C05450=1092.796,439.335,-104.729,178.655,25.944,154.047
C05451=1092.802,439.581,-104.773,178.657,25.957,154.050
C05452=1092.809,439.827,-104.817,178.661,25.970,154.053
C05453=1092.815,440.073,-104.861,178.665,25.983,154.056
C05454=1092.822,440.320,-104.905,178.667,25.995,154.059
C05455=1092.829,440.565,-104.948,178.671,26.009,154.062
C05456=1092.836,440.811,-104.992,178.674,26.022,154.065
C05457=1092.842,441.057,-105.036,178.677,26.035,154.068
C05458=1092.849,441.303,-105.080,178.680,26.048,154.071
C05459=1092.855,441.549,-105.124,178.684,26.061,154.074
C05460=1092.862,441.795,-105.168,178.687,26.074,154.077
C05461=1092.868,442.041,-105.212,178.690,26.088,154.080
C05462=1092.875,442.287,-105.256,178.693,26.101,154.083
C05463=1092.881,442.532,-105.299,178.697,26.115,154.086
C05464=1092.888,442.778,-105.344,178.700,26.128,154.089
C05465=1092.894,443.024,-105.388,178.703,26.142,154.092
C05466=1092.901,443.270,-105.432,178.707,26.155,154.095
C05467=1092.908,443.516,-105.477,178.710,26.169,154.098
C05468=1092.914,443.762,-105.521,178.713,26.182,154.101
C05469=1092.921,444.007,-105.565,178.716,26.196,154.104
C05470=1092.927,444.253,-105.610,178.719,26.210,154.107
C05471=1092.934,444.499,-105.654,178.723,26.224,154.110
C05472=1092.941,444.745,-105.698,178.725,26.237,154.114
C05473=1092.947,444.991,-105.743,178.728,26.251,154.117
C05474=1092.954,445.237,-105.787,178.730,26.265,154.120
C05475=1092.960,445.482,-105.831,178.733,26.279,154.123
C05476=1092.968,445.728,-105.876,178.735,26.292,154.126
C05477=1092.973,445.974,-105.921,178.737,26.306,154.130
C05478=1092.980,446.220,-105.965,178.738,26.319,154.133
C05479=1092.988,446.466,-106.010,178.741,26.333,154.136
C05480=1092.994,446.712,-106.054,178.741,26.347,154.140
C05481=1093.000,446.958,-106.099,178.743,26.361,154.143
C05482=1093.007,447.204,-106.144,178.744,26.374,154.146
C05483=1093.014,447.449,-106.189,178.745,26.388,154.150
C05484=1093.020,447.695,-106.233,178.746,26.401,154.153
C05485=1093.027,447.941,-106.278,178.747,26.415,154.156
C05486=1093.034,448.187,-106.323,178.747,26.429,154.160
C05487=1093.040,448.432,-106.368,178.747,26.442,154.163
C05488=1093.047,448.678,-106.413,178.748,26.456,154.166
C05489=1093.054,448.924,-106.457,178.748,26.469,154.170
C05490=1093.060,449.170,-106.503,178.748,26.483,154.173
C05491=1093.067,449.415,-106.547,178.747,26.496,154.177
C05492=1093.074,449.661,-106.592,178.748,26.510,154.180
C05493=1093.081,449.906,-106.637,178.748,26.523,154.184
C05494=1093.089,450.153,-106.681,178.747,26.535,154.187
C05495=1092.703,450.144,-106.858,178.697,26.740,154.244
C05496=1092.694,449.897,-106.813,178.697,26.727,154.241
C05497=1092.687,449.651,-106.768,178.698,26.714,154.237
C05498=1092.680,449.406,-106.724,178.698,26.700,154.234
C05499=1092.673,449.161,-106.679,178.698,26.686,154.230
C05500=1092.667,448.915,-106.634,178.698,26.673,154.227
C05501=1092.660,448.669,-106.589,178.698,26.660,154.224
C05502=1092.653,448.423,-106.544,178.697,26.646,154.220
C05503=1092.647,448.177,-106.499,178.697,26.633,154.217
C05504=1092.640,447.932,-106.454,178.697,26.619,154.213
C05505=1092.633,447.686,-106.409,178.695,26.605,154.210
C05506=1092.627,447.440,-106.364,178.695,26.591,154.207
C05507=1092.620,447.195,-106.320,178.694,26.578,154.203
C05508=1092.613,446.949,-106.275,178.692,26.564,154.200
C05509=1092.607,446.702,-106.230,178.691,26.550,154.197
C05510=1092.600,446.457,-106.186,178.689,26.536,154.193
C05511=1092.593,446.211,-106.141,178.687,26.523,154.190
C05512=1092.586,445.966,-106.096,178.686,26.509,154.187
C05513=1092.580,445.719,-106.052,178.684,26.495,154.183
C05514=1092.573,445.473,-106.007,178.682,26.482,154.180
C05515=1092.566,445.228,-105.962,178.679,26.468,154.177
C05516=1092.560,444.982,-105.918,178.677,26.454,154.174
C05517=1092.553,444.736,-105.874,178.674,26.440,154.170
C05518=1092.547,444.490,-105.828,178.671,26.427,154.167
C05519=1092.540,444.244,-105.785,178.668,26.413,154.164
C05520=1092.533,443.999,-105.740,178.664,26.399,154.161
C05521=1092.526,443.752,-105.696,178.661,26.385,154.158
C05522=1092.520,443.507,-105.651,178.658,26.371,154.155
C05523=1092.513,443.261,-105.607,178.655,26.358,154.152
C05524=1092.507,443.016,-105.563,178.651,26.344,154.149
C05525=1092.500,442.770,-105.519,178.647,26.330,154.146
C05526=1092.493,442.524,-105.474,178.644,26.317,154.143
C05527=1092.487,442.278,-105.431,178.641,26.303,154.139
C05528=1092.480,442.032,-105.386,178.638,26.290,154.136
C05529=1092.474,441.786,-105.342,178.634,26.276,154.133
C05530=1092.467,441.540,-105.298,178.631,26.263,154.130
C05531=1092.460,441.294,-105.254,178.628,26.250,154.127
C05532=1092.454,441.048,-105.210,178.624,26.237,154.125
C05533=1092.448,440.802,-105.166,178.621,26.224,154.122
C05534=1092.441,440.556,-105.122,178.618,26.210,154.119
C05535=1092.434,440.311,-105.078,178.614,26.197,154.116
C05536=1092.428,440.065,-105.034,178.611,26.185,154.113
C05537=1092.421,439.818,-104.990,178.608,26.171,154.110
C05538=1092.414,439.573,-104.947,178.604,26.158,154.107
C05539=1092.407,439.327,-104.903,178.601,26.146,154.104
C05540=1092.397,438.921,-104.831,178.596,26.124,154.099
C05541=1092.386,438.515,-104.759,178.590,26.104,154.095
C05542=1092.375,438.111,-104.687,178.585,26.083,154.090
C05543=1092.364,437.705,-104.616,178.579,26.062,154.086
C05544=1092.358,437.459,-104.572,178.576,26.050,154.083
C05545=1092.351,437.214,-104.529,178.573,26.037,154.080
C05546=1092.345,436.967,-104.486,178.570,26.025,154.077
C05547=1092.338,436.721,-104.442,178.566,26.012,154.075
C05548=1092.331,436.475,-104.398,178.562,25.999,154.072
C05549=1092.325,436.229,-104.355,178.560,25.987,154.069
C05550=1092.319,435.983,-104.311,178.556,25.975,154.066
C05551=1092.311,435.737,-104.268,178.553,25.963,154.064
C05552=1092.306,435.491,-104.225,178.550,25.951,154.061
C05553=1092.300,435.245,-104.182,178.546,25.938,154.058
C05554=1092.293,434.999,-104.139,178.544,25.927,154.056
C05555=1092.286,434.753,-104.095,178.540,25.914,154.053
C05556=1092.279,434.507,-104.053,178.537,25.902,154.050
C05557=1092.273,434.260,-104.010,178.533,25.890,154.048
C05558=1092.267,434.015,-103.966,178.530,25.878,154.045
C05559=1092.261,433.769,-103.924,178.527,25.866,154.042
C05560=1092.254,433.522,-103.880,178.524,25.854,154.040
C05561=1092.247,433.276,-103.837,178.521,25.843,154.037
C05562=1092.242,433.030,-103.794,178.517,25.831,154.035
C05563=1092.235,432.784,-103.752,178.514,25.819,154.032
C05564=1092.229,432.538,-103.709,178.510,25.807,154.029
C05565=1092.222,432.291,-103.666,178.508,25.796,154.027
C05566=1092.215,432.046,-103.623,178.505,25.784,154.024
C05567=1092.209,431.800,-103.580,178.501,25.772,154.022
C05568=1092.202,431.553,-103.538,178.498,25.761,154.019
C05569=1092.196,431.307,-103.494,178.495,25.750,154.017
C05570=1092.189,431.061,-103.452,178.491,25.738,154.014
C05571=1092.183,430.815,-103.410,178.488,25.726,154.012
C05572=1092.177,430.568,-103.367,178.485,25.716,154.010
C05573=1092.170,430.322,-103.324,178.481,25.704,154.007
C05574=1092.164,430.077,-103.282,178.478,25.692,154.005
C05575=1092.158,429.830,-103.239,178.475,25.681,154.002
C05576=1092.151,429.584,-103.196,178.472,25.670,154.000
C05577=1092.145,429.337,-103.155,178.469,25.659,153.997
C05578=1092.138,429.091,-103.112,178.466,25.648,153.995
C05579=1092.132,428.845,-103.069,178.463,25.637,153.993
C05580=1092.126,428.599,-103.027,178.459,25.625,153.990
C05581=1092.119,428.352,-102.985,178.456,25.614,153.988
C05582=1092.112,428.106,-102.943,178.453,25.603,153.985
C05583=1092.106,427.860,-102.900,178.449,25.593,153.983
C05584=1092.100,427.613,-102.859,178.447,25.582,153.981
C05585=1092.093,427.367,-102.815,178.443,25.571,153.978
C05586=1092.087,427.121,-102.773,178.440,25.560,153.976
C05587=1092.081,426.874,-102.731,178.437,25.549,153.974
C05588=1092.074,426.629,-102.689,178.433,25.539,153.972
C05589=1092.068,426.382,-102.647,178.430,25.528,153.969
C05590=1092.062,426.136,-102.605,178.427,25.518,153.967
C05591=1092.055,425.889,-102.563,178.423,25.507,153.965
C05592=1092.049,425.658,-102.524,178.421,25.497,153.963
C05593=1092.043,425.427,-102.485,178.418,25.487,153.961
C05594=1092.037,425.196,-102.445,178.415,25.477,153.958
C05595=1092.031,424.965,-102.406,178.411,25.467,153.956
C05596=1092.025,424.733,-102.366,178.409,25.457,153.954
C05597=1092.019,424.503,-102.327,178.406,25.447,153.952
C05598=1092.013,424.271,-102.287,178.403,25.437,153.950
C05599=1092.008,424.040,-102.249,178.399,25.427,153.948
C05600=1092.001,423.793,-102.206,178.396,25.417,153.946
C05601=1091.995,423.547,-102.165,178.393,25.407,153.944
C05602=1091.988,423.300,-102.123,178.390,25.396,153.941
C05603=1091.982,423.054,-102.082,178.387,25.386,153.939
C05604=1091.976,422.807,-102.040,178.384,25.376,153.937
C05605=1091.970,422.562,-101.998,178.381,25.366,153.935
C05606=1091.963,422.315,-101.956,178.377,25.356,153.933
C05607=1091.957,422.069,-101.914,178.374,25.345,153.931
C05608=1091.951,421.822,-101.873,178.371,25.335,153.929
C05609=1091.944,421.576,-101.832,178.368,25.325,153.926
C05610=1091.938,421.330,-101.790,178.365,25.316,153.924
C05611=1091.931,421.083,-101.748,178.362,25.305,153.922
C05612=1091.925,420.836,-101.707,178.358,25.295,153.920
C05613=1091.919,420.591,-101.666,178.355,25.286,153.918
C05614=1091.913,420.343,-101.625,178.352,25.275,153.916
C05615=1091.907,420.097,-101.584,178.349,25.266,153.914
C05616=1091.900,419.850,-101.542,178.345,25.256,153.912
C05617=1091.893,419.604,-101.501,178.342,25.246,153.910
C05618=1091.887,419.358,-101.459,178.339,25.236,153.908
C05619=1091.881,419.111,-101.418,178.336,25.227,153.906
C05620=1091.874,418.864,-101.377,178.334,25.217,153.904
C05621=1091.869,418.618,-101.336,178.330,25.208,153.902
C05622=1091.863,418.372,-101.295,178.327,25.198,153.900
C05623=1091.856,418.124,-101.253,178.324,25.188,153.898
C05624=1091.850,417.879,-101.213,178.321,25.179,153.896
C05625=1091.844,417.632,-101.171,178.317,25.169,153.894
C05626=1091.838,417.386,-101.130,178.314,25.159,153.892
C05627=1091.831,417.139,-101.089,178.311,25.150,153.890
C05628=1091.821,416.758,-101.026,178.306,25.135,153.887
C05629=1091.812,416.375,-100.962,178.301,25.120,153.884
C05630=1091.803,415.993,-100.899,178.296,25.106,153.881
C05631=1091.793,415.612,-100.835,178.292,25.092,153.878
C05632=1091.786,415.365,-100.795,178.288,25.082,153.876
C05633=1091.780,415.119,-100.755,178.286,25.074,153.874
C05634=1091.773,414.872,-100.713,178.282,25.064,153.873
C05635=1091.767,414.625,-100.673,178.279,25.055,153.871
C05636=1091.761,414.378,-100.632,178.276,25.046,153.869
C05637=1091.755,414.133,-100.591,178.273,25.037,153.867
C05638=1091.748,413.886,-100.551,178.270,25.028,153.865
C05639=1091.742,413.638,-100.510,178.267,25.018,153.863
C05640=1091.736,413.392,-100.470,178.263,25.010,153.861
C05641=1091.730,413.146,-100.429,178.261,25.001,153.860
C05642=1091.723,412.899,-100.388,178.258,24.992,153.858
C05643=1091.717,412.653,-100.348,178.254,24.983,153.856
C05644=1091.711,412.406,-100.308,178.251,24.973,153.854
C05645=1091.705,412.159,-100.267,178.248,24.965,153.852
C05646=1091.698,411.913,-100.227,178.245,24.956,153.851
C05647=1091.692,411.665,-100.186,178.242,24.947,153.849
C05648=1091.685,411.354,-100.135,178.238,24.936,153.847
C05649=1091.676,411.041,-100.084,178.234,24.925,153.844
C05650=1091.668,410.729,-100.033,178.230,24.914,153.842
C05651=1091.661,410.417,-99.983,178.226,24.903,153.840
C05652=1091.655,410.170,-99.942,178.223,24.894,153.838
C05653=1091.649,409.924,-99.902,178.221,24.885,153.836
C05654=1091.642,409.677,-99.862,178.217,24.877,153.835
C05655=1091.636,409.431,-99.821,178.214,24.868,153.833
C05656=1091.631,409.183,-99.781,178.211,24.860,153.831
C05657=1091.624,408.937,-99.741,178.208,24.851,153.829
C05658=1091.618,408.690,-99.701,178.205,24.842,153.828
C05659=1091.611,408.444,-99.661,178.202,24.834,153.826
C05660=1091.606,408.196,-99.621,178.198,24.825,153.824
C05661=1091.600,407.950,-99.581,178.196,24.817,153.823
C05662=1091.593,407.703,-99.541,178.192,24.808,153.821
C05663=1091.587,407.457,-99.500,178.190,24.800,153.819
C05664=1091.581,407.210,-99.461,178.186,24.791,153.818
C05665=1091.575,406.963,-99.421,178.184,24.783,153.816
C05666=1091.568,406.716,-99.381,178.180,24.775,153.814
C05667=1091.562,406.469,-99.341,178.177,24.767,153.813
C05668=1091.557,406.223,-99.301,178.174,24.758,153.811
C05669=1091.551,405.976,-99.261,178.171,24.750,153.809
C05670=1091.545,405.730,-99.221,178.168,24.742,153.808
C05671=1091.539,405.482,-99.182,178.165,24.734,153.806
C05672=1091.532,405.236,-99.142,178.162,24.725,153.805
C05673=1091.526,404.989,-99.102,178.159,24.718,153.803
C05674=1091.520,404.742,-99.063,178.156,24.709,153.801
C05675=1091.514,404.495,-99.023,178.153,24.701,153.800
C05676=1091.508,404.249,-98.984,178.149,24.693,153.798
C05677=1091.501,404.003,-98.944,178.147,24.685,153.797
C05678=1091.495,403.755,-98.905,178.143,24.677,153.795
C05679=1091.489,403.508,-98.865,178.141,24.669,153.794
C05680=1091.483,403.261,-98.826,178.138,24.661,153.792
C05681=1091.476,403.015,-98.786,178.134,24.653,153.791
C05682=1091.471,402.768,-98.747,178.132,24.645,153.789
C05683=1091.465,402.521,-98.707,178.128,24.637,153.787
C05684=1091.458,402.274,-98.668,178.125,24.630,153.786
C05685=1091.452,402.028,-98.628,178.123,24.622,153.784
C05686=1091.446,401.781,-98.589,178.119,24.614,153.783
C05687=1091.440,401.534,-98.550,178.116,24.606,153.781
C05688=1091.434,401.287,-98.510,178.113,24.598,153.780
C05689=1091.427,401.040,-98.471,178.110,24.591,153.778
C05690=1091.422,400.794,-98.432,178.107,24.583,153.777
C05691=1091.416,400.547,-98.393,178.104,24.575,153.775
C05692=1091.410,400.299,-98.353,178.101,24.568,153.774
C05693=1091.403,400.053,-98.315,178.098,24.560,153.772
C05694=1091.397,399.806,-98.276,178.095,24.552,153.771
C05695=1091.391,399.559,-98.236,178.092,24.544,153.769
C05696=1091.385,399.312,-98.197,178.089,24.537,153.768
C05697=1091.379,399.066,-98.158,178.086,24.529,153.767
C05698=1091.373,398.819,-98.119,178.083,24.522,153.765
C05699=1091.367,398.572,-98.079,178.080,24.514,153.764
C05700=1091.361,398.349,-98.044,178.077,24.508,153.762
C05701=1091.355,398.126,-98.009,178.074,24.500,153.761
C05702=1091.351,397.902,-97.974,178.071,24.494,153.760
C05703=1091.345,397.679,-97.939,178.069,24.487,153.759
C05704=1091.339,397.455,-97.903,178.066,24.480,153.757
C05705=1091.333,397.232,-97.868,178.063,24.474,153.756
C05706=1091.328,397.008,-97.834,178.060,24.467,153.755
C05707=1091.323,396.785,-97.798,178.058,24.461,153.753
C05708=1091.316,396.538,-97.759,178.055,24.453,153.752
C05709=1091.311,396.291,-97.721,178.052,24.446,153.751
C05710=1091.304,396.044,-97.682,178.049,24.438,153.749
C05711=1091.299,395.798,-97.643,178.046,24.431,153.748
C05712=1091.292,395.551,-97.605,178.043,24.424,153.747
C05713=1091.287,395.304,-97.566,178.040,24.417,153.745
C05714=1091.280,395.057,-97.527,178.037,24.409,153.744
C05715=1091.275,394.810,-97.488,178.034,24.402,153.742
C05716=1091.268,394.563,-97.450,178.030,24.395,153.741
C05717=1091.262,394.316,-97.411,178.028,24.388,153.740
C05718=1091.256,394.070,-97.372,178.025,24.380,153.738
C05719=1091.249,393.823,-97.334,178.022,24.373,153.737
C05720=1091.244,393.576,-97.295,178.019,24.367,153.736
C05721=1091.237,393.328,-97.257,178.015,24.359,153.734
C05722=1091.232,393.082,-97.218,178.012,24.352,153.733
C05723=1091.226,392.835,-97.180,178.009,24.345,153.732
C05724=1091.219,392.588,-97.141,178.007,24.338,153.730
C05725=1091.214,392.341,-97.103,178.004,24.331,153.729
C05726=1091.207,392.094,-97.064,178.001,24.324,153.728
C05727=1091.201,391.848,-97.026,177.997,24.317,153.727
C05728=1091.195,391.600,-96.988,177.994,24.310,153.725
C05729=1091.189,391.354,-96.949,177.991,24.303,153.724
C05730=1091.183,391.106,-96.911,177.988,24.296,153.723
C05731=1091.177,390.860,-96.873,177.985,24.290,153.722
C05732=1091.171,390.613,-96.835,177.982,24.283,153.720
C05733=1091.164,390.366,-96.797,177.979,24.275,153.719
C05734=1091.158,390.119,-96.759,177.976,24.269,153.718
C05735=1091.152,389.872,-96.721,177.973,24.262,153.717
C05736=1091.147,389.625,-96.683,177.970,24.255,153.715
C05737=1091.140,389.379,-96.644,177.967,24.249,153.714
C05738=1091.134,389.131,-96.606,177.964,24.242,153.713
C05739=1091.128,388.884,-96.568,177.961,24.235,153.712
C05740=1091.122,388.638,-96.530,177.957,24.228,153.710
C05741=1091.116,388.390,-96.492,177.954,24.222,153.709
C05742=1091.110,388.143,-96.455,177.951,24.215,153.708
C05743=1091.104,387.897,-96.417,177.948,24.208,153.707
C05744=1091.098,387.650,-96.379,177.945,24.202,153.706
C05745=1091.091,387.403,-96.341,177.943,24.195,153.704
C05746=1091.086,387.156,-96.303,177.939,24.189,153.703
C05747=1091.080,386.909,-96.265,177.937,24.182,153.702
C05748=1091.074,386.662,-96.227,177.934,24.175,153.701
C05749=1091.068,386.415,-96.189,177.931,24.169,153.700
C05750=1091.062,386.168,-96.151,177.927,24.162,153.699
C05751=1091.056,385.921,-96.113,177.924,24.156,153.697
C05752=1091.050,385.674,-96.076,177.921,24.149,153.696
C05753=1091.044,385.427,-96.038,177.918,24.143,153.695
C05754=1091.038,385.180,-96.000,177.915,24.136,153.694
C05755=1091.032,384.933,-95.962,177.912,24.130,153.693
C05756=1091.026,384.716,-95.929,177.910,24.124,153.692
C05757=1091.021,384.500,-95.897,177.906,24.118,153.691
C05758=1091.016,384.282,-95.863,177.904,24.113,153.690
C05759=1091.011,384.066,-95.831,177.901,24.107,153.689
C05760=1091.005,383.849,-95.797,177.898,24.101,153.688
C05761=1091.000,383.633,-95.764,177.896,24.095,153.687
C05762=1090.995,383.416,-95.731,177.893,24.090,153.686
C05763=1090.991,383.199,-95.698,177.891,24.084,153.685
C05764=1090.985,382.952,-95.661,177.888,24.078,153.684
C05765=1090.978,382.705,-95.624,177.885,24.072,153.682
C05766=1090.972,382.458,-95.586,177.882,24.065,153.681
C05767=1090.966,382.211,-95.548,177.879,24.059,153.680
C05768=1090.960,381.964,-95.511,177.875,24.053,153.679
C05769=1090.954,381.717,-95.473,177.872,24.047,153.678
C05770=1090.948,381.470,-95.437,177.869,24.040,153.677
C05771=1090.942,381.223,-95.399,177.866,24.034,153.676
C05772=1090.937,380.976,-95.362,177.863,24.028,153.675
C05773=1090.930,380.729,-95.325,177.860,24.022,153.674
C05774=1090.924,380.481,-95.288,177.857,24.016,153.673
C05775=1090.918,380.234,-95.250,177.854,24.010,153.672
C05776=1090.912,379.987,-95.213,177.851,24.003,153.671
C05777=1090.906,379.741,-95.176,177.848,23.997,153.670
C05778=1090.900,379.493,-95.139,177.845,23.991,153.669
C05779=1090.894,379.246,-95.102,177.842,23.985,153.667
C05780=1090.888,378.999,-95.064,177.839,23.979,153.666
C05781=1090.882,378.752,-95.027,177.835,23.973,153.665
C05782=1090.877,378.505,-94.990,177.832,23.967,153.664
C05783=1090.870,378.258,-94.953,177.829,23.961,153.663
C05784=1090.864,378.011,-94.916,177.827,23.955,153.662
C05785=1090.859,377.764,-94.879,177.824,23.949,153.661
C05786=1090.852,377.517,-94.843,177.821,23.943,153.660
C05787=1090.846,377.270,-94.805,177.818,23.937,153.659
C05788=1090.840,377.023,-94.769,177.814,23.931,153.658
C05789=1090.835,376.775,-94.731,177.811,23.925,153.657
C05790=1090.829,376.528,-94.694,177.808,23.919,153.656
C05791=1090.823,376.281,-94.658,177.805,23.913,153.655
C05792=1090.817,376.034,-94.620,177.802,23.907,153.654
C05793=1090.811,375.787,-94.583,177.799,23.901,153.653
C05794=1090.805,375.540,-94.547,177.796,23.895,153.652
C05795=1090.799,375.292,-94.510,177.793,23.890,153.651
C05796=1090.793,375.045,-94.473,177.790,23.884,153.650
C05797=1090.787,374.798,-94.436,177.787,23.878,153.649
C05798=1090.781,374.551,-94.400,177.784,23.872,153.648
C05799=1090.775,374.304,-94.363,177.781,23.866,153.647
C05800=1090.769,374.057,-94.326,177.778,23.860,153.646
C05801=1090.763,373.809,-94.289,177.774,23.855,153.645
C05802=1090.758,373.563,-94.253,177.771,23.849,153.644
C05803=1090.752,373.315,-94.216,177.769,23.843,153.643
C05804=1090.746,373.068,-94.180,177.766,23.837,153.642
C05805=1090.740,372.821,-94.144,177.763,23.832,153.641
C05806=1090.734,372.573,-94.107,177.759,23.826,153.641
C05807=1090.728,372.326,-94.070,177.756,23.820,153.640
C05808=1090.721,372.079,-94.034,177.753,23.814,153.639
C05809=1090.716,371.832,-93.997,177.750,23.809,153.638
C05810=1090.710,371.584,-93.961,177.747,23.804,153.637
C05811=1090.703,371.337,-93.925,177.744,23.798,153.636
C05812=1090.694,370.932,-93.865,177.739,23.789,153.634
C05813=1090.684,370.525,-93.805,177.734,23.779,153.633
C05814=1090.675,370.119,-93.745,177.729,23.770,153.631
C05815=1090.665,369.714,-93.686,177.724,23.761,153.630
C05816=1090.659,369.467,-93.650,177.721,23.756,153.629
C05817=1090.652,369.220,-93.613,177.718,23.750,153.628
C05818=1090.647,368.972,-93.577,177.715,23.744,153.627
C05819=1090.641,368.725,-93.541,177.712,23.739,153.626
C05820=1090.635,368.478,-93.505,177.708,23.734,153.626
C05821=1090.629,368.231,-93.469,177.706,23.728,153.625
C05822=1090.624,367.983,-93.432,177.703,23.723,153.624
C05823=1090.618,367.736,-93.396,177.699,23.717,153.623
C05824=1090.612,367.489,-93.361,177.696,23.712,153.622
C05825=1090.605,367.242,-93.324,177.693,23.706,153.621
C05826=1090.600,366.994,-93.288,177.691,23.701,153.620
C05827=1090.594,366.747,-93.252,177.687,23.696,153.619
C05828=1090.588,366.500,-93.216,177.684,23.690,153.618
C05829=1090.582,366.252,-93.180,177.681,23.684,153.618
C05830=1090.577,366.006,-93.144,177.678,23.679,153.617
C05831=1090.571,365.758,-93.108,177.675,23.674,153.616
C05832=1090.565,365.510,-93.072,177.672,23.669,153.615
C05833=1090.559,365.263,-93.036,177.668,23.663,153.614
C05834=1090.553,365.016,-93.000,177.666,23.658,153.613
C05835=1090.547,364.768,-92.965,177.663,23.653,153.613
C05836=1090.541,364.521,-92.929,177.659,23.647,153.612
C05837=1090.535,364.273,-92.892,177.657,23.642,153.611
C05838=1090.530,364.027,-92.857,177.654,23.637,153.610
C05839=1090.524,363.779,-92.821,177.650,23.632,153.609
C05840=1090.518,363.531,-92.786,177.647,23.627,153.609
C05841=1090.512,363.284,-92.750,177.645,23.622,153.608
C05842=1090.506,363.037,-92.714,177.641,23.616,153.607
C05843=1090.500,362.789,-92.678,177.638,23.611,153.606
C05844=1090.494,362.543,-92.643,177.636,23.606,153.605
C05845=1090.488,362.295,-92.608,177.632,23.601,153.604
C05846=1090.482,362.047,-92.572,177.629,23.595,153.604
C05847=1090.476,361.800,-92.536,177.625,23.590,153.603
C05848=1090.470,361.553,-92.501,177.623,23.585,153.602
C05849=1090.464,361.305,-92.465,177.620,23.580,153.601
C05850=1090.459,361.058,-92.430,177.616,23.575,153.601
C05851=1090.453,360.810,-92.394,177.614,23.570,153.600
C05852=1090.447,360.563,-92.359,177.611,23.565,153.599
C05853=1090.441,360.316,-92.323,177.607,23.560,153.598
C05854=1090.434,360.068,-92.288,177.605,23.555,153.597
C05855=1090.429,359.821,-92.252,177.601,23.550,153.597
C05856=1090.423,359.574,-92.217,177.598,23.545,153.596
C05857=1090.418,359.327,-92.181,177.596,23.540,153.595
C05858=1090.412,359.079,-92.146,177.592,23.535,153.594
C05859=1090.405,358.831,-92.111,177.589,23.530,153.594
C05860=1090.400,358.584,-92.076,177.586,23.525,153.593
C05861=1090.394,358.337,-92.040,177.583,23.520,153.592
C05862=1090.388,358.090,-92.005,177.579,23.515,153.591
C05863=1090.381,357.842,-91.969,177.577,23.510,153.591
C05864=1090.373,357.451,-91.914,177.571,23.502,153.590
C05865=1090.363,357.062,-91.859,177.567,23.494,153.588
C05866=1090.355,356.671,-91.803,177.562,23.486,153.587
C05867=1090.345,356.280,-91.748,177.558,23.479,153.586
C05868=1090.340,356.033,-91.713,177.554,23.474,153.585
C05869=1090.333,355.785,-91.678,177.551,23.469,153.585
C05870=1090.327,355.538,-91.642,177.548,23.464,153.584
C05871=1090.322,355.290,-91.607,177.545,23.459,153.583
C05872=1090.315,355.043,-91.573,177.542,23.454,153.582
C05873=1090.310,354.795,-91.538,177.539,23.449,153.582
C05874=1090.304,354.548,-91.502,177.536,23.444,153.581
C05875=1090.298,354.300,-91.468,177.533,23.440,153.580
C05876=1090.292,354.053,-91.432,177.530,23.435,153.580
C05877=1090.286,353.805,-91.398,177.527,23.430,153.579
C05878=1090.281,353.558,-91.363,177.524,23.425,153.578
C05879=1090.275,353.310,-91.328,177.520,23.420,153.577
C05880=1090.269,353.063,-91.293,177.518,23.416,153.577
C05881=1090.263,352.816,-91.258,177.514,23.411,153.576
C05882=1090.257,352.568,-91.223,177.512,23.407,153.575
C05883=1090.252,352.321,-91.188,177.508,23.402,153.575
C05884=1090.245,352.073,-91.154,177.505,23.397,153.574
C05885=1090.240,351.826,-91.119,177.502,23.392,153.573
C05886=1090.233,351.578,-91.084,177.499,23.387,153.573
C05887=1090.227,351.331,-91.050,177.496,23.383,153.572
C05888=1090.222,351.084,-91.015,177.493,23.378,153.571
C05889=1090.216,350.836,-90.980,177.490,23.374,153.571
C05890=1090.210,350.588,-90.946,177.487,23.369,153.570
C05891=1090.204,350.340,-90.911,177.484,23.364,153.569
C05892=1090.198,350.093,-90.876,177.481,23.360,153.569
C05893=1090.193,349.846,-90.842,177.477,23.355,153.568
C05894=1090.186,349.598,-90.808,177.475,23.350,153.567
C05895=1090.181,349.350,-90.773,177.471,23.346,153.567
C05896=1090.175,349.103,-90.739,177.469,23.341,153.566
C05897=1090.169,348.855,-90.704,177.465,23.337,153.566
C05898=1090.164,348.607,-90.670,177.462,23.332,153.565
C05899=1090.157,348.361,-90.635,177.459,23.327,153.564
C05900=1090.152,348.112,-90.600,177.456,23.323,153.564
C05901=1090.146,347.865,-90.566,177.453,23.318,153.563
C05902=1090.140,347.618,-90.532,177.450,23.314,153.562
C05903=1090.135,347.370,-90.497,177.447,23.309,153.562
C05904=1090.128,347.122,-90.463,177.444,23.305,153.561
C05905=1090.123,346.875,-90.429,177.441,23.300,153.560
C05906=1090.117,346.628,-90.395,177.438,23.296,153.560
C05907=1090.111,346.379,-90.360,177.434,23.291,153.559
C05908=1090.105,346.132,-90.326,177.432,23.287,153.559
C05909=1090.099,345.885,-90.292,177.428,23.282,153.558
C05910=1090.094,345.637,-90.257,177.426,23.278,153.557
C05911=1090.088,345.389,-90.223,177.422,23.273,153.557
C05912=1090.082,345.141,-90.189,177.420,23.269,153.556
C05913=1090.076,344.894,-90.155,177.416,23.264,153.555
C05914=1090.070,344.647,-90.121,177.413,23.260,153.555
C05915=1090.065,344.398,-90.086,177.410,23.255,153.554
C05916=1090.055,344.010,-90.033,177.405,23.248,153.553
C05917=1090.046,343.623,-89.980,177.400,23.241,153.552
C05918=1090.037,343.235,-89.926,177.395,23.234,153.551
C05919=1090.028,342.847,-89.874,177.391,23.228,153.551
C05920=1090.022,342.600,-89.840,177.388,23.223,153.550
C05921=1090.016,342.353,-89.805,177.384,23.219,153.549
C05922=1090.011,342.105,-89.772,177.382,23.215,153.549
C05923=1090.004,341.857,-89.738,177.379,23.211,153.548
C05924=1089.998,341.610,-89.704,177.375,23.206,153.548
C05925=1089.993,341.362,-89.670,177.373,23.202,153.547
C05926=1089.987,341.114,-89.636,177.369,23.197,153.547
C05927=1089.981,340.866,-89.603,177.366,23.193,153.546
C05928=1089.975,340.619,-89.569,177.363,23.189,153.545
C05929=1089.970,340.372,-89.535,177.360,23.185,153.545
C05930=1089.963,340.123,-89.501,177.357,23.180,153.544
C05931=1089.958,339.876,-89.467,177.354,23.176,153.544
C05932=1089.952,339.628,-89.434,177.351,23.172,153.543
C05933=1089.946,339.381,-89.400,177.348,23.167,153.543
C05934=1089.941,339.133,-89.366,177.345,23.163,153.542
C05935=1089.935,338.886,-89.332,177.342,23.159,153.541
C05936=1089.929,338.638,-89.299,177.339,23.155,153.541
C05937=1089.924,338.390,-89.266,177.336,23.151,153.540
C05938=1089.918,338.142,-89.232,177.332,23.146,153.540
C05939=1089.912,337.895,-89.198,177.330,23.142,153.539
C05940=1089.906,337.647,-89.164,177.326,23.138,153.539
C05941=1089.900,337.399,-89.130,177.323,23.134,153.538
C05942=1089.894,337.151,-89.098,177.321,23.130,153.538
C05943=1089.888,336.904,-89.064,177.317,23.125,153.537
C05944=1089.882,336.656,-89.030,177.314,23.122,153.537
C05945=1089.877,336.408,-88.997,177.311,23.117,153.536
C05946=1089.871,336.160,-88.964,177.308,23.113,153.535
C05947=1089.865,335.913,-88.930,177.305,23.109,153.535
C05948=1089.859,335.665,-88.897,177.302,23.105,153.534
C05949=1089.854,335.417,-88.864,177.299,23.101,153.534
C05950=1089.848,335.169,-88.830,177.296,23.097,153.533
C05951=1089.842,334.922,-88.796,177.293,23.092,153.533
C05952=1089.836,334.675,-88.763,177.290,23.088,153.532
C05953=1089.830,334.427,-88.730,177.287,23.085,153.532
C05954=1089.825,334.179,-88.697,177.284,23.080,153.531
C05955=1089.819,333.931,-88.663,177.281,23.076,153.531
C05956=1089.813,333.683,-88.631,177.277,23.072,153.530
C05957=1089.807,333.435,-88.597,177.275,23.068,153.530
C05958=1089.802,333.187,-88.564,177.272,23.064,153.529
C05959=1089.795,332.940,-88.530,177.268,23.059,153.529
C05960=1089.790,332.693,-88.497,177.265,23.056,153.528
C05961=1089.784,332.445,-88.464,177.263,23.052,153.528
C05962=1089.779,332.197,-88.430,177.259,23.047,153.527
C05963=1089.772,331.949,-88.398,177.256,23.043,153.527
C05964=1089.767,331.701,-88.364,177.253,23.040,153.526
C05965=1089.761,331.454,-88.332,177.250,23.036,153.526
C05966=1089.755,331.206,-88.298,177.247,23.032,153.525
C05967=1089.749,330.958,-88.266,177.244,23.028,153.525
C05968=1089.740,330.564,-88.213,177.239,23.022,153.524
C05969=1089.730,330.170,-88.161,177.234,23.015,153.523
C05970=1089.720,329.777,-88.110,177.229,23.009,153.523
C05971=1089.711,329.383,-88.056,177.224,23.003,153.522
C05972=1089.706,329.136,-88.025,177.221,22.999,153.521
C05973=1089.700,328.888,-87.991,177.219,22.995,153.521
C05974=1089.694,328.640,-87.959,177.216,22.992,153.521
C05975=1089.688,328.392,-87.925,177.212,22.987,153.520
C05976=1089.682,328.145,-87.893,177.209,22.984,153.520
C05977=1089.676,327.897,-87.861,177.206,22.980,153.519
C05978=1089.671,327.649,-87.827,177.203,22.976,153.519
C05979=1089.664,327.401,-87.794,177.200,22.972,153.518
C05980=1089.658,327.153,-87.762,177.197,22.968,153.518
C05981=1089.653,326.906,-87.729,177.194,22.965,153.517
C05982=1089.647,326.658,-87.697,177.191,22.960,153.517
C05983=1089.642,326.410,-87.664,177.188,22.957,153.516
C05984=1089.636,326.162,-87.631,177.185,22.953,153.516
C05985=1089.629,325.914,-87.599,177.182,22.949,153.516
C05986=1089.624,325.666,-87.566,177.178,22.945,153.515
C05987=1089.618,325.419,-87.534,177.176,22.942,153.515
C05988=1089.612,325.171,-87.502,177.173,22.938,153.514
C05989=1089.606,324.923,-87.469,177.170,22.934,153.514
C05990=1089.601,324.675,-87.436,177.166,22.930,153.513
C05991=1089.594,324.427,-87.403,177.163,22.926,153.513
C05992=1089.589,324.180,-87.371,177.161,22.923,153.513
C05993=1089.584,323.932,-87.338,177.158,22.919,153.512
C05994=1089.578,323.683,-87.306,177.154,22.914,153.512
C05995=1089.571,323.436,-87.274,177.151,22.911,153.511
C05996=1089.567,323.188,-87.241,177.149,22.908,153.511
C05997=1089.560,322.940,-87.209,177.146,22.904,153.510
C05998=1089.554,322.692,-87.177,177.142,22.900,153.510
C05999=1089.549,322.445,-87.144,177.139,22.896,153.510
C06000=1089.543,322.197,-87.112,177.136,22.892,153.509
C06001=1089.537,321.949,-87.080,177.134,22.889,153.509
C06002=1089.531,321.701,-87.047,177.131,22.885,153.508
C06003=1089.526,321.453,-87.015,177.127,22.881,153.508
C06004=1089.520,321.205,-86.983,177.124,22.877,153.507
C06005=1089.514,320.957,-86.950,177.121,22.874,153.507
C06006=1089.509,320.710,-86.918,177.119,22.870,153.506
C06007=1089.503,320.462,-86.886,177.116,22.866,153.506
C06008=1089.497,320.215,-86.854,177.112,22.862,153.506
C06009=1089.492,319.966,-86.821,177.109,22.858,153.505
C06010=1089.486,319.718,-86.789,177.106,22.855,153.505
C06011=1089.481,319.470,-86.758,177.103,22.852,153.504
C06012=1089.475,319.222,-86.725,177.101,22.848,153.504
C06013=1089.469,318.975,-86.693,177.097,22.844,153.504
C06014=1089.463,318.727,-86.661,177.094,22.840,153.503
C06015=1089.458,318.479,-86.628,177.091,22.836,153.503
C06016=1089.452,318.231,-86.597,177.088,22.833,153.502
C06017=1089.446,317.983,-86.565,177.085,22.829,153.502
C06018=1089.441,317.735,-86.533,177.082,22.825,153.502
C06019=1089.435,317.487,-86.501,177.079,22.822,153.501
C06020=1089.426,317.087,-86.449,177.074,22.816,153.500
C06021=1089.417,316.686,-86.398,177.070,22.810,153.500
C06022=1089.408,316.286,-86.345,177.065,22.804,153.499
C06023=1089.398,315.885,-86.294,177.060,22.798,153.498
C06024=1089.393,315.638,-86.262,177.057,22.794,153.498
C06025=1089.388,315.390,-86.231,177.054,22.791,153.498
C06026=1089.382,315.142,-86.199,177.051,22.787,153.497
C06027=1089.376,314.894,-86.167,177.048,22.783,153.497
C06028=1089.370,314.646,-86.135,177.044,22.780,153.497
C06029=1089.364,314.398,-86.103,177.041,22.776,153.496
C06030=1089.358,314.151,-86.072,177.039,22.773,153.496
C06031=1089.352,313.902,-86.041,177.036,22.770,153.495
C06032=1089.347,313.654,-86.009,177.033,22.766,153.495
C06033=1089.341,313.406,-85.977,177.030,22.763,153.495
C06034=1089.334,313.158,-85.946,177.027,22.759,153.494
C06035=1089.329,312.911,-85.914,177.023,22.755,153.494
C06036=1089.323,312.663,-85.882,177.020,22.752,153.494
C06037=1089.317,312.415,-85.852,177.017,22.748,153.493
C06038=1089.311,312.167,-85.820,177.014,22.745,153.493
C06039=1089.306,311.919,-85.788,177.012,22.741,153.493
C06040=1089.300,311.671,-85.756,177.009,22.738,153.492
C06041=1089.294,311.423,-85.725,177.006,22.735,153.492
C06042=1089.288,311.175,-85.693,177.003,22.731,153.491
C06043=1089.283,310.927,-85.662,176.999,22.728,153.491
C06044=1089.276,310.679,-85.631,176.996,22.724,153.491
C06045=1089.271,310.431,-85.599,176.993,22.721,153.490
C06046=1089.265,310.184,-85.568,176.990,22.717,153.490
C06047=1089.259,309.935,-85.537,176.987,22.714,153.490
C06048=1089.254,309.688,-85.505,176.984,22.711,153.489
C06049=1089.247,309.440,-85.474,176.981,22.707,153.489
C06050=1089.242,309.192,-85.443,176.978,22.704,153.489
C06051=1089.236,308.943,-85.411,176.976,22.700,153.488
C06052=1089.230,308.696,-85.381,176.972,22.697,153.488
C06053=1089.225,308.448,-85.349,176.969,22.693,153.488
C06054=1089.219,308.200,-85.317,176.966,22.690,153.487
C06055=1089.213,307.952,-85.287,176.963,22.687,153.487
C06056=1089.207,307.705,-85.255,176.960,22.683,153.487
C06057=1089.201,307.456,-85.224,176.957,22.680,153.486
C06058=1089.196,307.209,-85.193,176.954,22.676,153.486
C06059=1089.190,306.961,-85.162,176.951,22.673,153.486
C06060=1089.184,306.712,-85.131,176.948,22.670,153.485
C06061=1089.179,306.464,-85.099,176.945,22.666,153.485
C06062=1089.173,306.217,-85.069,176.942,22.663,153.485
C06063=1089.167,305.968,-85.037,176.939,22.659,153.484
C06064=1089.161,305.720,-85.006,176.936,22.656,153.484
C06065=1089.156,305.473,-84.975,176.933,22.652,153.484
C06066=1089.149,305.224,-84.944,176.930,22.649,153.483
C06067=1089.144,304.976,-84.913,176.927,22.646,153.483
C06068=1089.138,304.729,-84.882,176.924,22.643,153.483
C06069=1089.133,304.481,-84.851,176.921,22.639,153.482
C06070=1089.127,304.232,-84.820,176.918,22.636,153.482
C06071=1089.121,303.985,-84.789,176.915,22.633,153.482
C06072=1089.112,303.587,-84.740,176.910,22.627,153.481
C06073=1089.104,303.189,-84.690,176.906,22.622,153.481
C06074=1089.094,302.791,-84.641,176.901,22.616,153.480
C06075=1089.085,302.394,-84.591,176.895,22.610,153.480
C06076=1089.080,302.145,-84.560,176.892,22.607,153.479
C06077=1089.074,301.898,-84.530,176.889,22.604,153.479
C06078=1089.068,301.650,-84.498,176.886,22.601,153.479
C06079=1089.063,301.402,-84.468,176.884,22.597,153.478
C06080=1089.058,301.154,-84.437,176.881,22.594,153.478
C06081=1089.051,300.906,-84.406,176.878,22.590,153.478
C06082=1089.045,300.658,-84.376,176.875,22.587,153.477
C06083=1089.040,300.410,-84.345,176.872,22.584,153.477
C06084=1089.034,300.162,-84.315,176.869,22.581,153.477
C06085=1089.029,299.914,-84.284,176.866,22.577,153.476
C06086=1089.024,299.666,-84.253,176.863,22.574,153.476
C06087=1089.018,299.418,-84.222,176.860,22.571,153.476
C06088=1089.013,299.170,-84.192,176.857,22.567,153.475
C06089=1089.007,298.922,-84.162,176.854,22.564,153.475
C06090=1089.001,298.673,-84.130,176.851,22.561,153.475
C06091=1088.995,298.425,-84.100,176.848,22.557,153.474
C06092=1088.990,298.178,-84.070,176.845,22.554,153.474
C06093=1088.984,297.929,-84.039,176.842,22.551,153.474
C06094=1088.979,297.682,-84.008,176.839,22.547,153.474
C06095=1088.973,297.434,-83.978,176.836,22.544,153.473
C06096=1088.967,297.186,-83.948,176.834,22.541,153.473
C06097=1088.962,296.938,-83.917,176.831,22.538,153.473
C06098=1088.956,296.689,-83.887,176.827,22.535,153.472
C06099=1088.950,296.441,-83.856,176.824,22.532,153.472
C06100=1088.944,296.193,-83.826,176.821,22.528,153.472
C06101=1088.938,295.945,-83.796,176.818,22.525,153.472
C06102=1088.933,295.697,-83.765,176.816,22.522,153.471
C06103=1088.927,295.449,-83.736,176.813,22.519,153.471
C06104=1088.921,295.201,-83.705,176.810,22.515,153.471
C06105=1088.916,294.953,-83.674,176.807,22.512,153.470
C06106=1088.910,294.705,-83.644,176.804,22.509,153.470
C06107=1088.905,294.457,-83.614,176.801,22.506,153.470
C06108=1088.899,294.209,-83.584,176.798,22.502,153.470
C06109=1088.893,293.961,-83.554,176.795,22.500,153.469
C06110=1088.888,293.713,-83.524,176.792,22.496,153.469
C06111=1088.882,293.465,-83.494,176.789,22.493,153.469
C06112=1088.876,293.217,-83.463,176.786,22.490,153.468
C06113=1088.870,292.968,-83.433,176.783,22.487,153.468
C06114=1088.864,292.720,-83.403,176.780,22.483,153.468
C06115=1088.858,292.472,-83.373,176.777,22.480,153.468
C06116=1088.853,292.224,-83.343,176.774,22.477,153.467
C06117=1088.847,291.976,-83.313,176.771,22.474,153.467
C06118=1088.841,291.728,-83.283,176.768,22.471,153.467
C06119=1088.836,291.480,-83.253,176.765,22.468,153.467
C06120=1088.830,291.231,-83.223,176.762,22.464,153.466
C06121=1088.824,290.984,-83.193,176.759,22.462,153.466
C06122=1088.819,290.735,-83.163,176.756,22.458,153.466
C06123=1088.814,290.488,-83.133,176.753,22.455,153.465
C06124=1088.804,290.104,-83.087,176.748,22.450,153.465
C06125=1088.796,289.720,-83.041,176.744,22.445,153.465
C06126=1088.787,289.337,-82.995,176.739,22.441,153.464
C06127=1088.777,288.953,-82.948,176.735,22.436,153.464
C06128=1088.772,288.704,-82.919,176.732,22.433,153.464
C06129=1088.766,288.456,-82.889,176.729,22.430,153.463
C06130=1088.760,288.208,-82.859,176.726,22.427,153.463
C06131=1088.754,287.960,-82.830,176.723,22.424,153.463
C06132=1088.749,287.712,-82.800,176.720,22.421,153.463
C06133=1088.743,287.464,-82.770,176.717,22.418,153.462
C06134=1088.738,287.216,-82.740,176.714,22.414,153.462
C06135=1088.732,286.968,-82.711,176.711,22.412,153.462
C06136=1088.726,286.720,-82.681,176.708,22.408,153.462
C06137=1088.721,286.472,-82.651,176.705,22.405,153.461
C06138=1088.715,286.223,-82.622,176.702,22.402,153.461
C06139=1088.709,285.975,-82.593,176.699,22.399,153.461
C06140=1088.703,285.727,-82.563,176.696,22.396,153.461
C06141=1088.698,285.479,-82.533,176.693,22.393,153.460
C06142=1088.692,285.230,-82.503,176.690,22.390,153.460
C06143=1088.686,284.983,-82.474,176.688,22.387,153.460
C06144=1088.681,284.734,-82.445,176.684,22.384,153.460
C06145=1088.675,284.486,-82.415,176.681,22.381,153.459
C06146=1088.669,284.238,-82.386,176.678,22.378,153.459
C06147=1088.664,283.989,-82.356,176.675,22.375,153.459
C06148=1088.658,283.742,-82.326,176.672,22.372,153.459
C06149=1088.651,283.493,-82.297,176.669,22.368,153.458
C06150=1088.647,283.246,-82.268,176.666,22.366,153.458
C06151=1088.641,282.997,-82.238,176.663,22.362,153.458
C06152=1088.636,282.749,-82.208,176.661,22.359,153.458
C06153=1088.629,282.501,-82.179,176.658,22.357,153.457
C06154=1088.624,282.252,-82.150,176.655,22.353,153.457
C06155=1088.618,282.005,-82.121,176.652,22.351,153.457
C06156=1088.613,281.756,-82.091,176.649,22.347,153.457
C06157=1088.607,281.508,-82.062,176.646,22.344,153.456
C06158=1088.601,281.260,-82.033,176.643,22.341,153.456
C06159=1088.596,281.012,-82.004,176.640,22.338,153.456
C06160=1088.590,280.763,-81.975,176.637,22.335,153.456
C06161=1088.585,280.515,-81.946,176.635,22.332,153.455
C06162=1088.578,280.267,-81.917,176.632,22.330,153.455
C06163=1088.573,280.018,-81.887,176.629,22.326,153.455
C06164=1088.567,279.771,-81.858,176.626,22.324,153.455
C06165=1088.562,279.522,-81.829,176.623,22.320,153.455
C06166=1088.555,279.274,-81.800,176.620,22.317,153.454
C06167=1088.550,279.025,-81.771,176.617,22.314,153.454
C06168=1088.544,278.778,-81.742,176.614,22.311,153.454
C06169=1088.539,278.529,-81.712,176.611,22.309,153.454
C06170=1088.533,278.281,-81.683,176.608,22.305,153.453
C06171=1088.527,278.033,-81.654,176.605,22.303,153.453
C06172=1088.522,277.785,-81.626,176.602,22.299,153.453
C06173=1088.516,277.536,-81.596,176.599,22.297,153.453
C06174=1088.510,277.288,-81.567,176.596,22.293,153.452
C06175=1088.506,277.040,-81.538,176.593,22.291,153.452
C06176=1088.496,276.665,-81.495,176.590,22.286,153.452
C06177=1088.488,276.291,-81.452,176.585,22.282,153.452
C06178=1088.479,275.917,-81.408,176.580,22.278,153.451
C06179=1088.470,275.543,-81.365,176.576,22.273,153.451
C06180=1088.465,275.295,-81.335,176.573,22.270,153.451
C06181=1088.459,275.047,-81.306,176.570,22.267,153.450
C06182=1088.453,274.799,-81.278,176.567,22.264,153.450
C06183=1088.448,274.550,-81.248,176.565,22.261,153.450
C06184=1088.442,274.302,-81.220,176.561,22.258,153.450
C06185=1088.436,274.054,-81.191,176.558,22.255,153.450
C06186=1088.431,273.805,-81.162,176.555,22.252,153.449
C06187=1088.425,273.557,-81.134,176.552,22.250,153.449
C06188=1088.419,273.309,-81.105,176.550,22.247,153.449
C06189=1088.414,273.060,-81.076,176.547,22.244,153.449
C06190=1088.409,272.812,-81.048,176.544,22.241,153.448
C06191=1088.402,272.564,-81.019,176.541,22.238,153.448
C06192=1088.396,272.315,-80.991,176.538,22.235,153.448
C06193=1088.391,272.067,-80.963,176.535,22.232,153.448
C06194=1088.386,271.819,-80.933,176.533,22.230,153.448
C06195=1088.380,271.571,-80.905,176.530,22.226,153.447
C06196=1088.374,271.323,-80.876,176.527,22.223,153.447
C06197=1088.368,271.074,-80.848,176.523,22.221,153.447
C06198=1088.363,270.826,-80.820,176.520,22.217,153.447
C06199=1088.357,270.577,-80.790,176.517,22.215,153.447
C06200=1088.352,270.329,-80.762,176.515,22.212,153.446
C06201=1088.346,270.081,-80.734,176.512,22.209,153.446
C06202=1088.341,269.832,-80.706,176.509,22.206,153.446
C06203=1088.334,269.584,-80.677,176.506,22.203,153.446
C06204=1088.328,269.336,-80.648,176.503,22.200,153.446
C06205=1088.323,269.088,-80.620,176.501,22.198,153.445
C06206=1088.317,268.839,-80.592,176.498,22.195,153.445
C06207=1088.311,268.591,-80.563,176.495,22.192,153.445
C06208=1088.305,268.343,-80.535,176.492,22.189,153.445
C06209=1088.300,268.095,-80.507,176.488,22.186,153.445
C06210=1088.295,267.846,-80.478,176.486,22.183,153.444
C06211=1088.290,267.597,-80.450,176.483,22.181,153.444
C06212=1088.283,267.349,-80.421,176.480,22.178,153.444
C06213=1088.278,267.101,-80.393,176.477,22.174,153.444
C06214=1088.272,266.853,-80.365,176.474,22.172,153.444
C06215=1088.267,266.604,-80.337,176.472,22.169,153.443
C06216=1088.261,266.356,-80.309,176.469,22.167,153.443
C06217=1088.255,266.108,-80.281,176.466,22.163,153.443
C06218=1088.249,265.859,-80.252,176.463,22.160,153.443
C06219=1088.244,265.611,-80.224,176.460,22.158,153.443
C06220=1088.238,265.362,-80.196,176.457,22.155,153.442
C06221=1088.233,265.114,-80.168,176.454,22.152,153.442
C06222=1088.227,264.865,-80.140,176.451,22.149,153.442
C06223=1088.222,264.617,-80.112,176.448,22.146,153.442
C06224=1088.216,264.369,-80.084,176.446,22.144,153.442
C06225=1088.210,264.121,-80.056,176.443,22.141,153.441
C06226=1088.204,263.872,-80.028,176.440,22.138,153.441
C06227=1088.198,263.624,-80.000,176.437,22.135,153.441
C06228=1088.190,263.253,-79.958,176.433,22.131,153.441
C06229=1088.180,262.881,-79.916,176.428,22.127,153.441
C06230=1088.172,262.510,-79.874,176.424,22.123,153.440
C06231=1088.164,262.139,-79.833,176.420,22.119,153.440
C06232=1088.157,261.890,-79.805,176.417,22.116,153.440
C06233=1088.152,261.642,-79.777,176.414,22.113,153.440
C06234=1088.146,261.393,-79.749,176.412,22.110,153.439
C06235=1088.140,261.145,-79.722,176.408,22.108,153.439
C06236=1088.134,260.896,-79.694,176.405,22.105,153.439
C06237=1088.129,260.648,-79.666,176.402,22.102,153.439
C06238=1088.124,260.400,-79.638,176.400,22.100,153.439
C06239=1088.117,260.151,-79.611,176.397,22.097,153.439
C06240=1088.112,259.903,-79.583,176.394,22.094,153.439
C06241=1088.106,259.654,-79.555,176.391,22.091,153.438
C06242=1088.100,259.407,-79.527,176.389,22.088,153.438
C06243=1088.095,259.158,-79.500,176.385,22.086,153.438
C06244=1088.089,258.909,-79.472,176.382,22.083,153.438
C06245=1088.083,258.661,-79.444,176.379,22.080,153.438
C06246=1088.077,258.412,-79.417,176.377,22.078,153.437
C06247=1088.072,258.164,-79.389,176.374,22.075,153.437
C06248=1088.066,257.916,-79.361,176.371,22.072,153.437
C06249=1088.060,257.667,-79.334,176.368,22.069,153.437
C06250=1088.054,257.419,-79.306,176.366,22.067,153.437
C06251=1088.049,257.170,-79.279,176.362,22.064,153.437
C06252=1088.043,256.922,-79.251,176.359,22.061,153.436
C06253=1088.037,256.673,-79.224,176.357,22.059,153.436
C06254=1088.032,256.425,-79.196,176.354,22.056,153.436
C06255=1088.025,256.177,-79.169,176.351,22.052,153.436
C06256=1088.020,255.928,-79.141,176.348,22.050,153.436
C06257=1088.015,255.680,-79.113,176.346,22.047,153.435
C06258=1088.009,255.432,-79.087,176.343,22.045,153.435
C06259=1088.003,255.182,-79.059,176.339,22.042,153.435
C06260=1087.997,254.935,-79.032,176.337,22.039,153.435
C06261=1087.992,254.686,-79.004,176.334,22.037,153.435
C06262=1087.987,254.438,-78.977,176.331,22.033,153.435
C06263=1087.981,254.189,-78.950,176.328,22.030,153.434
C06264=1087.975,253.941,-78.922,176.326,22.028,153.434
C06265=1087.969,253.692,-78.895,176.323,22.025,153.434
C06266=1087.964,253.444,-78.868,176.320,22.022,153.434
C06267=1087.958,253.195,-78.840,176.317,22.020,153.434
C06268=1087.953,252.947,-78.813,176.314,22.017,153.433
C06269=1087.947,252.698,-78.786,176.311,22.014,153.433
C06270=1087.942,252.450,-78.758,176.309,22.012,153.433
C06271=1087.936,252.202,-78.731,176.306,22.009,153.433
C06272=1087.930,251.953,-78.704,176.303,22.006,153.433
C06273=1087.924,251.705,-78.676,176.300,22.003,153.433
C06274=1087.919,251.456,-78.649,176.298,22.000,153.432
C06275=1087.913,251.208,-78.623,176.295,21.998,153.432
C06276=1087.908,250.959,-78.595,176.291,21.995,153.432
C06277=1087.902,250.711,-78.568,176.289,21.992,153.432
C06278=1087.897,250.462,-78.540,176.286,21.990,153.432
C06279=1087.891,250.214,-78.514,176.283,21.986,153.432
C06280=1087.883,249.839,-78.473,176.279,21.983,153.431
C06281=1087.875,249.466,-78.432,176.275,21.978,153.431
C06282=1087.866,249.091,-78.391,176.271,21.975,153.431
C06283=1087.857,248.717,-78.350,176.266,21.970,153.430
C06284=1087.852,248.468,-78.323,176.264,21.968,153.430
C06285=1087.847,248.220,-78.297,176.261,21.965,153.430
C06286=1087.842,247.971,-78.269,176.258,21.962,153.430
C06287=1087.836,247.723,-78.243,176.255,21.959,153.430
C06288=1087.831,247.474,-78.215,176.253,21.956,153.430
C06289=1087.825,247.226,-78.189,176.250,21.953,153.429
C06290=1087.819,246.977,-78.162,176.248,21.951,153.429
C06291=1087.814,246.728,-78.135,176.244,21.948,153.429
C06292=1087.808,246.480,-78.108,176.241,21.946,153.429
C06293=1087.802,246.232,-78.081,176.239,21.943,153.429
C06294=1087.796,245.983,-78.055,176.236,21.940,153.429
C06295=1087.791,245.734,-78.027,176.233,21.938,153.428
C06296=1087.785,245.486,-78.001,176.231,21.935,153.428
C06297=1087.780,245.238,-77.974,176.227,21.932,153.428
C06298=1087.774,244.989,-77.947,176.225,21.929,153.428
C06299=1087.769,244.741,-77.920,176.222,21.927,153.428
C06300=1087.763,244.492,-77.893,176.219,21.924,153.428
C06301=1087.757,244.244,-77.867,176.216,21.921,153.427
C06302=1087.752,243.996,-77.840,176.214,21.919,153.427
C06303=1087.746,243.747,-77.814,176.211,21.916,153.427
C06304=1087.741,243.498,-77.787,176.208,21.913,153.427
C06305=1087.735,243.250,-77.760,176.205,21.911,153.427
C06306=1087.730,243.001,-77.734,176.202,21.908,153.427
C06307=1087.723,242.752,-77.707,176.200,21.906,153.426
C06308=1087.718,242.503,-77.681,176.197,21.903,153.426
C06309=1087.712,242.255,-77.654,176.194,21.900,153.426
C06310=1087.706,242.007,-77.627,176.192,21.898,153.426
C06311=1087.700,241.758,-77.601,176.189,21.895,153.426
C06312=1087.695,241.510,-77.574,176.185,21.892,153.426
C06313=1087.689,241.261,-77.548,176.183,21.890,153.426
C06314=1087.683,241.012,-77.522,176.180,21.887,153.425
C06315=1087.678,240.764,-77.495,176.178,21.884,153.425
C06316=1087.672,240.515,-77.469,176.175,21.882,153.425
C06317=1087.667,240.266,-77.442,176.172,21.879,153.425
C06318=1087.661,240.018,-77.415,176.169,21.876,153.425
C06319=1087.656,239.769,-77.389,176.166,21.874,153.425
C06320=1087.649,239.521,-77.363,176.163,21.871,153.425
C06321=1087.644,239.273,-77.336,176.161,21.868,153.424
C06322=1087.638,239.024,-77.311,176.158,21.866,153.424
C06323=1087.632,238.775,-77.284,176.156,21.863,153.424
C06324=1087.627,238.527,-77.258,176.153,21.860,153.424
C06325=1087.622,238.279,-77.232,176.149,21.858,153.424
C06326=1087.616,238.030,-77.206,176.147,21.855,153.424
C06327=1087.610,237.781,-77.179,176.144,21.852,153.423
C06328=1087.605,237.533,-77.152,176.142,21.850,153.423
C06329=1087.599,237.284,-77.127,176.139,21.847,153.423
C06330=1087.593,237.036,-77.100,176.136,21.844,153.423
C06331=1087.588,236.787,-77.074,176.133,21.842,153.423
C06332=1087.580,236.406,-77.034,176.129,21.837,153.422
C06333=1087.570,236.025,-76.994,176.125,21.834,153.422
C06334=1087.562,235.644,-76.954,176.121,21.829,153.422
C06335=1087.553,235.263,-76.914,176.117,21.826,153.422
C06336=1087.548,235.014,-76.888,176.114,21.823,153.422
C06337=1087.542,234.765,-76.861,176.111,21.820,153.421
C06338=1087.537,234.517,-76.835,176.108,21.818,153.421
C06339=1087.531,234.268,-76.809,176.106,21.815,153.421
C06340=1087.525,234.019,-76.783,176.103,21.812,153.421
C06341=1087.520,233.771,-76.758,176.100,21.810,153.421
C06342=1087.514,233.522,-76.732,176.098,21.807,153.421
C06343=1087.509,233.274,-76.705,176.095,21.804,153.421
C06344=1087.503,233.025,-76.679,176.092,21.802,153.420
C06345=1087.497,232.776,-76.654,176.089,21.799,153.420
C06346=1087.492,232.527,-76.628,176.087,21.797,153.420
C06347=1087.486,232.279,-76.601,176.084,21.794,153.420
C06348=1087.481,232.031,-76.576,176.081,21.791,153.420
C06349=1087.475,231.782,-76.550,176.079,21.789,153.420
C06350=1087.469,231.533,-76.524,176.076,21.786,153.419
C06351=1087.463,231.285,-76.498,176.073,21.784,153.419
C06352=1087.459,231.036,-76.472,176.070,21.781,153.419
C06353=1087.452,230.788,-76.447,176.068,21.778,153.419
C06354=1087.447,230.539,-76.421,176.065,21.776,153.419
C06355=1087.441,230.290,-76.395,176.063,21.773,153.419
C06356=1087.435,230.041,-76.370,176.060,21.770,153.419
C06357=1087.430,229.793,-76.343,176.057,21.768,153.418
C06358=1087.424,229.545,-76.318,176.054,21.765,153.418
C06359=1087.418,229.296,-76.292,176.051,21.762,153.418
C06360=1087.413,229.047,-76.266,176.049,21.760,153.418
C06361=1087.407,228.798,-76.241,176.046,21.758,153.418
C06362=1087.402,228.550,-76.215,176.043,21.755,153.418
C06363=1087.396,228.301,-76.190,176.040,21.752,153.418
C06364=1087.390,228.052,-76.164,176.038,21.750,153.417
C06365=1087.384,227.803,-76.139,176.035,21.747,153.417
C06366=1087.379,227.555,-76.113,176.033,21.745,153.417
C06367=1087.373,227.307,-76.088,176.030,21.742,153.417
C06368=1087.367,227.058,-76.062,176.027,21.740,153.417
C06369=1087.361,226.809,-76.036,176.024,21.737,153.417
C06370=1087.356,226.561,-76.011,176.021,21.734,153.417
C06371=1087.350,226.312,-75.986,176.019,21.732,153.416
C06372=1087.345,226.063,-75.960,176.016,21.729,153.416
C06373=1087.340,225.815,-75.934,176.014,21.726,153.416
C06374=1087.334,225.566,-75.909,176.011,21.724,153.416
C06375=1087.328,225.317,-75.883,176.008,21.721,153.416
C06376=1087.323,225.069,-75.858,176.005,21.718,153.416
C06377=1087.316,224.820,-75.832,176.003,21.716,153.415
C06378=1087.311,224.571,-75.807,176.000,21.713,153.415
C06379=1087.306,224.323,-75.782,175.998,21.711,153.415
C06380=1087.300,224.074,-75.756,175.995,21.708,153.415
C06381=1087.294,223.825,-75.731,175.993,21.706,153.415
C06382=1087.289,223.577,-75.705,175.989,21.703,153.415
C06383=1087.283,223.328,-75.680,175.987,21.701,153.415
C06384=1087.274,222.938,-75.641,175.983,21.696,153.414
C06385=1087.266,222.549,-75.601,175.979,21.692,153.414
C06386=1087.257,222.159,-75.561,175.974,21.688,153.414
C06387=1087.249,221.769,-75.522,175.970,21.684,153.414
C06388=1087.243,221.520,-75.497,175.967,21.682,153.414
C06389=1087.236,221.272,-75.472,175.965,21.679,153.413
C06390=1087.232,221.023,-75.446,175.962,21.676,153.413
C06391=1087.226,220.774,-75.421,175.960,21.675,153.413
C06392=1087.219,220.525,-75.396,175.956,21.672,153.413
C06393=1087.214,220.277,-75.371,175.954,21.669,153.413
C06394=1087.209,220.028,-75.346,175.951,21.666,153.413
C06395=1087.203,219.780,-75.321,175.949,21.664,153.413
C06396=1087.197,219.531,-75.296,175.946,21.661,153.412
C06397=1087.191,219.282,-75.271,175.944,21.659,153.412
C06398=1087.186,219.034,-75.245,175.941,21.656,153.412
C06399=1087.180,218.784,-75.221,175.938,21.654,153.412
C06400=1087.175,218.536,-75.196,175.935,21.651,153.412
C06401=1087.169,218.287,-75.171,175.933,21.648,153.412
C06402=1087.164,218.039,-75.146,175.931,21.647,153.412
C06403=1087.158,217.790,-75.121,175.928,21.644,153.412
C06404=1087.152,217.542,-75.096,175.925,21.641,153.411
C06405=1087.146,217.292,-75.071,175.922,21.639,153.411
C06406=1087.140,217.044,-75.046,175.920,21.636,153.411
C06407=1087.135,216.795,-75.022,175.917,21.633,153.411
C06408=1087.129,216.546,-74.996,175.915,21.631,153.411
C06409=1087.124,216.297,-74.972,175.912,21.628,153.411
C06410=1087.118,216.049,-74.946,175.909,21.626,153.410
C06411=1087.113,215.800,-74.922,175.906,21.623,153.410
C06412=1087.107,215.552,-74.897,175.904,21.621,153.410
C06413=1087.101,215.303,-74.872,175.901,21.618,153.410
C06414=1087.097,215.054,-74.848,175.899,21.615,153.410
C06415=1087.090,214.805,-74.822,175.897,21.613,153.410
C06416=1087.085,214.557,-74.798,175.894,21.610,153.410
C06417=1087.079,214.308,-74.773,175.891,21.608,153.409
C06418=1087.074,214.060,-74.748,175.888,21.605,153.409
C06419=1087.068,213.810,-74.724,175.886,21.602,153.409
C06420=1087.062,213.562,-74.700,175.883,21.600,153.409
C06421=1087.057,213.313,-74.674,175.881,21.597,153.409
C06422=1087.052,213.064,-74.649,175.877,21.595,153.409
C06423=1087.046,212.816,-74.625,175.875,21.593,153.409
C06424=1087.040,212.567,-74.600,175.873,21.590,153.408
C06425=1087.035,212.318,-74.576,175.870,21.587,153.408
C06426=1087.029,212.069,-74.551,175.868,21.585,153.408
C06427=1087.024,211.820,-74.527,175.865,21.582,153.408
C06428=1087.017,211.572,-74.501,175.862,21.580,153.408
C06429=1087.012,211.323,-74.477,175.859,21.577,153.408
C06430=1087.007,211.075,-74.453,175.857,21.575,153.408
C06431=1087.001,210.825,-74.428,175.854,21.572,153.407
C06432=1086.995,210.577,-74.405,175.852,21.569,153.407
C06433=1086.989,210.328,-74.380,175.849,21.567,153.407
C06434=1086.983,210.080,-74.355,175.846,21.565,153.407
C06435=1086.978,209.831,-74.331,175.844,21.562,153.407
C06436=1086.969,209.445,-74.293,175.839,21.558,153.407
C06437=1086.961,209.059,-74.255,175.836,21.554,153.407
C06438=1086.952,208.674,-74.217,175.832,21.550,153.406
C06439=1086.944,208.287,-74.179,175.828,21.547,153.406
C06440=1086.920,207.262,-74.081,175.750,21.506,153.410
C06441=1086.914,207.012,-74.056,175.748,21.504,153.410
C06442=1086.909,206.764,-74.032,175.745,21.503,153.410
C06443=1086.903,206.515,-74.009,175.742,21.501,153.410
C06444=1086.898,206.266,-73.985,175.739,21.500,153.410
C06445=1086.893,206.018,-73.961,175.737,21.498,153.410
C06446=1086.886,205.769,-73.937,175.734,21.497,153.410
C06447=1086.881,205.519,-73.913,175.731,21.495,153.410
C06448=1086.875,205.271,-73.890,175.729,21.493,153.410
C06449=1086.870,205.023,-73.865,175.726,21.491,153.410
C06450=1086.865,204.773,-73.842,175.723,21.490,153.410
C06451=1086.859,204.525,-73.818,175.720,21.488,153.410
C06452=1086.854,204.276,-73.795,175.718,21.487,153.410
C06453=1086.847,204.027,-73.771,175.715,21.485,153.411
C06454=1086.842,203.778,-73.746,175.713,21.483,153.411
C06455=1086.837,203.529,-73.723,175.709,21.482,153.411
C06456=1086.831,203.281,-73.699,175.707,21.480,153.411
C06457=1086.826,203.032,-73.676,175.704,21.478,153.411
C06458=1086.820,202.783,-73.652,175.702,21.477,153.411
C06459=1086.815,202.534,-73.628,175.699,21.476,153.411
C06460=1086.809,202.286,-73.605,175.697,21.474,153.411
C06461=1086.803,202.036,-73.581,175.694,21.472,153.411
C06462=1086.797,201.788,-73.557,175.691,21.470,153.411
C06463=1086.791,201.539,-73.534,175.688,21.469,153.411
C06464=1086.786,201.290,-73.510,175.686,21.467,153.411
C06465=1086.780,201.041,-73.487,175.683,21.466,153.411
C06466=1086.775,200.793,-73.463,175.680,21.464,153.412
C06467=1086.769,200.544,-73.440,175.678,21.463,153.412
C06468=1086.763,200.295,-73.416,175.675,21.461,153.412
C06469=1086.758,200.046,-73.392,175.673,21.460,153.412
C06470=1086.752,199.797,-73.369,175.669,21.458,153.412
C06471=1086.746,199.549,-73.346,175.667,21.456,153.412
C06472=1086.741,199.299,-73.322,175.664,21.455,153.412
C06473=1086.735,199.051,-73.298,175.662,21.453,153.412
C06474=1086.729,198.802,-73.275,175.659,21.452,153.412
C06475=1086.724,198.553,-73.252,175.656,21.450,153.412
C06476=1086.718,198.305,-73.228,175.654,21.449,153.412
C06477=1086.712,198.056,-73.205,175.651,21.447,153.412
C06478=1086.707,197.807,-73.182,175.649,21.446,153.413
C06479=1086.701,197.557,-73.158,175.645,21.443,153.413
C06480=1086.695,197.309,-73.135,175.643,21.442,153.413
C06481=1086.689,197.060,-73.112,175.640,21.441,153.413
C06482=1086.684,196.811,-73.088,175.638,21.439,153.413
C06483=1086.678,196.562,-73.065,175.635,21.437,153.413
C06484=1086.672,196.313,-73.042,175.633,21.436,153.413
C06485=1086.667,196.064,-73.018,175.630,21.434,153.413
C06486=1086.662,195.815,-72.995,175.628,21.433,153.413
C06487=1086.656,195.567,-72.972,175.625,21.431,153.413
C06488=1086.650,195.318,-72.949,175.622,21.429,153.413
C06489=1086.645,195.069,-72.925,175.619,21.428,153.413
C06490=1086.639,194.820,-72.902,175.616,21.426,153.413
C06491=1086.634,194.571,-72.879,175.614,21.424,153.413
C06492=1086.629,194.322,-72.856,175.611,21.423,153.414
C06493=1086.623,194.074,-72.832,175.609,21.421,153.414
C06494=1086.617,193.825,-72.809,175.606,21.420,153.414
C06495=1086.611,193.576,-72.786,175.604,21.418,153.414
C06496=1086.606,193.328,-72.763,175.601,21.417,153.414
C06497=1086.601,193.078,-72.740,175.599,21.415,153.414
C06498=1086.595,192.830,-72.717,175.596,21.414,153.414
C06499=1086.589,192.581,-72.694,175.594,21.412,153.414
C06500=1086.584,192.332,-72.671,175.591,21.410,153.414
C06501=1086.578,192.054,-72.645,175.588,21.408,153.414
C06502=1086.571,191.776,-72.619,175.585,21.407,153.414
C06503=1086.565,191.498,-72.593,175.582,21.405,153.414
C06504=1086.559,191.220,-72.568,175.579,21.403,153.414
C06505=1086.553,190.971,-72.545,175.577,21.401,153.414
C06506=1086.548,190.722,-72.521,175.574,21.399,153.414
C06507=1086.543,190.474,-72.499,175.572,21.398,153.415
C06508=1086.537,190.225,-72.476,175.569,21.397,153.415
C06509=1086.531,189.976,-72.453,175.567,21.395,153.415
C06510=1086.526,189.727,-72.430,175.564,21.393,153.415
C06511=1086.521,189.478,-72.406,175.562,21.392,153.415
C06512=1086.515,189.229,-72.383,175.558,21.390,153.415
C06513=1086.509,188.980,-72.360,175.556,21.388,153.415
C06514=1086.504,188.732,-72.338,175.553,21.386,153.415
C06515=1086.498,188.483,-72.315,175.550,21.385,153.415
C06516=1086.493,188.234,-72.293,175.548,21.383,153.415
C06517=1086.488,187.984,-72.269,175.545,21.382,153.415
C06518=1086.482,187.735,-72.246,175.543,21.380,153.415
C06519=1086.477,187.487,-72.223,175.540,21.378,153.415
C06520=1086.471,187.238,-72.201,175.538,21.377,153.415
C06521=1086.466,186.989,-72.178,175.535,21.375,153.415
C06522=1086.460,186.741,-72.155,175.533,21.373,153.415
C06523=1086.455,186.491,-72.133,175.530,21.372,153.415
C06524=1086.449,186.243,-72.110,175.528,21.370,153.415
C06525=1086.444,185.994,-72.086,175.525,21.369,153.416
C06526=1086.439,185.745,-72.064,175.523,21.367,153.416
C06527=1086.433,185.495,-72.041,175.520,21.365,153.416
C06528=1086.428,185.246,-72.018,175.518,21.363,153.416
C06529=1086.422,184.998,-71.996,175.515,21.362,153.416
C06530=1086.417,184.749,-71.973,175.513,21.360,153.416
C06531=1086.411,184.500,-71.951,175.510,21.359,153.416
C06532=1086.405,184.251,-71.928,175.508,21.357,153.416
C06533=1086.399,184.002,-71.905,175.505,21.356,153.416
C06534=1086.393,183.753,-71.882,175.503,21.354,153.416
C06535=1086.387,183.504,-71.861,175.500,21.353,153.416
C06536=1086.382,183.256,-71.838,175.497,21.351,153.416
C06537=1086.376,183.007,-71.815,175.495,21.349,153.416
C06538=1086.371,182.757,-71.793,175.492,21.348,153.416
C06539=1086.364,182.509,-71.771,175.490,21.347,153.416
C06540=1086.359,182.260,-71.748,175.487,21.345,153.416
C06541=1086.353,182.010,-71.725,175.485,21.343,153.417
C06542=1086.348,181.762,-71.703,175.482,21.342,153.417
C06543=1086.342,181.513,-71.681,175.480,21.340,153.417
C06544=1086.336,181.264,-71.658,175.477,21.339,153.417
C06545=1086.331,181.015,-71.635,175.475,21.337,153.417
C06546=1086.324,180.766,-71.614,175.472,21.335,153.417
C06547=1086.319,180.518,-71.591,175.470,21.334,153.417
C06548=1086.314,180.268,-71.569,175.467,21.333,153.417
C06549=1086.308,180.019,-71.546,175.464,21.331,153.417
C06550=1086.302,179.770,-71.524,175.462,21.329,153.417
C06551=1086.296,179.521,-71.501,175.459,21.327,153.417
C06552=1086.291,179.273,-71.479,175.457,21.326,153.417
C06553=1086.285,179.024,-71.457,175.454,21.325,153.417
C06554=1086.279,178.774,-71.435,175.452,21.323,153.417
C06555=1086.274,178.526,-71.412,175.449,21.321,153.418
C06556=1086.268,178.277,-71.391,175.447,21.320,153.418
C06557=1086.262,178.028,-71.368,175.444,21.318,153.418
C06558=1086.257,177.779,-71.346,175.442,21.317,153.418
C06559=1086.251,177.530,-71.324,175.439,21.315,153.418
C06560=1086.246,177.281,-71.301,175.437,21.313,153.418
C06561=1086.240,177.032,-71.279,175.434,21.312,153.418
C06562=1086.234,176.783,-71.257,175.432,21.311,153.418
C06563=1086.229,176.534,-71.235,175.430,21.309,153.418
C06564=1086.223,176.285,-71.213,175.427,21.307,153.418
C06565=1086.216,176.007,-71.188,175.424,21.305,153.418
C06566=1086.210,175.729,-71.163,175.422,21.304,153.418
C06567=1086.204,175.451,-71.138,175.419,21.302,153.418
C06568=1086.198,175.173,-71.114,175.416,21.300,153.418
C06569=1086.193,174.923,-71.091,175.414,21.298,153.418
C06570=1086.186,174.674,-71.070,175.411,21.297,153.418
C06571=1086.181,174.426,-71.047,175.409,21.295,153.418
C06572=1086.176,174.177,-71.025,175.406,21.294,153.418
C06573=1086.170,173.928,-71.004,175.404,21.292,153.418
C06574=1086.165,173.678,-70.981,175.401,21.290,153.419
C06575=1086.158,173.430,-70.959,175.399,21.289,153.419
C06576=1086.154,173.181,-70.937,175.396,21.287,153.419
C06577=1086.147,172.932,-70.916,175.394,21.285,153.419
C06578=1086.142,172.682,-70.893,175.391,21.284,153.419
C06579=1086.137,172.434,-70.871,175.389,21.282,153.419
C06580=1086.131,172.185,-70.849,175.386,21.281,153.419
C06581=1086.126,171.936,-70.827,175.384,21.279,153.419
C06582=1086.120,171.687,-70.806,175.381,21.277,153.419
C06583=1086.115,171.438,-70.784,175.379,21.275,153.419
C06584=1086.109,171.189,-70.762,175.377,21.274,153.419
C06585=1086.103,170.940,-70.739,175.375,21.273,153.419
C06586=1086.098,170.691,-70.717,175.372,21.271,153.419
C06587=1086.092,170.442,-70.696,175.370,21.269,153.419
C06588=1086.087,170.193,-70.674,175.367,21.267,153.419
C06589=1086.081,169.944,-70.652,175.365,21.266,153.419
C06590=1086.076,169.695,-70.630,175.362,21.264,153.419
C06591=1086.070,169.446,-70.609,175.360,21.262,153.419
C06592=1086.065,169.197,-70.587,175.357,21.261,153.419
C06593=1086.059,168.948,-70.565,175.355,21.259,153.419
C06594=1086.054,168.699,-70.543,175.352,21.258,153.419
C06595=1086.048,168.451,-70.521,175.351,21.256,153.419
C06596=1086.043,168.202,-70.499,175.348,21.254,153.419
C06597=1086.037,167.953,-70.478,175.346,21.253,153.419
C06598=1086.032,167.704,-70.456,175.343,21.251,153.419
C06599=1086.026,167.454,-70.434,175.341,21.249,153.419
C06600=1086.021,167.206,-70.412,175.338,21.248,153.420
C06601=1086.015,166.956,-70.391,175.336,21.246,153.420
C06602=1086.010,166.708,-70.369,175.334,21.244,153.420
C06603=1086.004,166.458,-70.347,175.331,21.242,153.420
C06604=1085.999,166.209,-70.326,175.329,21.241,153.420
C06605=1085.993,165.960,-70.304,175.327,21.239,153.420
C06606=1085.988,165.711,-70.283,175.324,21.238,153.420
C06607=1085.983,165.462,-70.261,175.322,21.236,153.420
C06608=1085.977,165.213,-70.239,175.320,21.234,153.420
C06609=1085.972,164.964,-70.218,175.317,21.233,153.420
C06610=1085.966,164.715,-70.196,175.315,21.231,153.420
C06611=1085.961,164.466,-70.174,175.312,21.229,153.420
C06612=1085.955,164.217,-70.152,175.310,21.227,153.420
C06613=1085.950,163.968,-70.131,175.308,21.226,153.420
C06614=1085.944,163.719,-70.110,175.306,21.224,153.420
C06615=1085.938,163.470,-70.088,175.303,21.222,153.420
C06616=1085.934,163.221,-70.067,175.301,21.221,153.420
C06617=1085.928,162.973,-70.045,175.298,21.219,153.420
C06618=1085.923,162.723,-70.023,175.296,21.217,153.420
C06619=1085.917,162.474,-70.003,175.293,21.215,153.420
C06620=1085.912,162.225,-69.980,175.291,21.214,153.420
C06621=1085.906,161.976,-69.959,175.289,21.212,153.420
C06622=1085.901,161.728,-69.938,175.287,21.210,153.420
C06623=1085.896,161.477,-69.916,175.285,21.208,153.420
C06624=1085.890,161.229,-69.895,175.282,21.207,153.420
C06625=1085.884,160.980,-69.873,175.280,21.205,153.420
C06626=1085.878,160.731,-69.852,175.277,21.203,153.420
C06627=1085.873,160.482,-69.832,175.274,21.202,153.420
C06628=1085.867,160.233,-69.810,175.273,21.200,153.420
C06629=1085.861,159.954,-69.786,175.270,21.198,153.420
C06630=1085.855,159.676,-69.763,175.267,21.197,153.420
C06631=1085.848,159.398,-69.738,175.265,21.195,153.420
C06632=1085.842,159.119,-69.714,175.262,21.193,153.420
C06633=1085.837,158.870,-69.694,175.260,21.192,153.420
C06634=1085.831,158.620,-69.672,175.257,21.190,153.420
C06635=1085.826,158.372,-69.650,175.255,21.188,153.420
C06636=1085.820,158.123,-69.630,175.253,21.187,153.420
C06637=1085.814,157.873,-69.608,175.251,21.185,153.420
C06638=1085.809,157.625,-69.587,175.248,21.183,153.420
C06639=1085.803,157.376,-69.566,175.246,21.182,153.420
C06640=1085.797,157.127,-69.545,175.243,21.180,153.420
C06641=1085.792,156.877,-69.524,175.241,21.178,153.420
C06642=1085.786,156.629,-69.503,175.239,21.176,153.420
C06643=1085.780,156.379,-69.482,175.237,21.175,153.421
C06644=1085.776,156.130,-69.460,175.234,21.173,153.420
C06645=1085.770,155.881,-69.439,175.232,21.171,153.420
C06646=1085.764,155.632,-69.418,175.229,21.170,153.421
C06647=1085.759,155.383,-69.397,175.227,21.168,153.421
C06648=1085.753,155.134,-69.376,175.225,21.166,153.421
C06649=1085.748,154.885,-69.355,175.223,21.165,153.421
C06650=1085.742,154.636,-69.334,175.220,21.163,153.421
C06651=1085.737,154.387,-69.313,175.218,21.161,153.421
C06652=1085.731,154.138,-69.292,175.216,21.159,153.421
C06653=1085.725,153.889,-69.271,175.214,21.158,153.421
C06654=1085.720,153.640,-69.250,175.211,21.157,153.421
C06655=1085.713,153.391,-69.230,175.209,21.155,153.421
C06656=1085.708,153.142,-69.208,175.207,21.153,153.421
C06657=1085.702,152.893,-69.188,175.204,21.151,153.421
C06658=1085.696,152.643,-69.167,175.202,21.149,153.421
C06659=1085.691,152.395,-69.146,175.200,21.148,153.421
C06660=1085.686,152.145,-69.125,175.198,21.146,153.421
C06661=1085.680,151.897,-69.104,175.195,21.145,153.421
C06662=1085.674,151.647,-69.083,175.193,21.143,153.421
C06663=1085.669,151.398,-69.062,175.190,21.141,153.421
C06664=1085.663,151.150,-69.041,175.189,21.139,153.421
C06665=1085.658,150.900,-69.020,175.186,21.138,153.421
C06666=1085.652,150.651,-68.999,175.184,21.136,153.421
C06667=1085.647,150.402,-68.978,175.181,21.134,153.421
C06668=1085.641,150.153,-68.958,175.180,21.133,153.421
C06669=1085.635,149.904,-68.938,175.177,21.131,153.421
C06670=1085.630,149.654,-68.917,175.175,21.129,153.421
C06671=1085.624,149.406,-68.895,175.172,21.128,153.421
C06672=1085.619,149.157,-68.875,175.170,21.126,153.421
C06673=1085.614,148.908,-68.854,175.169,21.124,153.421
C06674=1085.608,148.658,-68.833,175.166,21.122,153.421
C06675=1085.602,148.409,-68.812,175.164,21.121,153.421
C06676=1085.596,148.160,-68.792,175.161,21.119,153.421
C06677=1085.591,147.911,-68.772,175.159,21.117,153.421
C06678=1085.586,147.662,-68.751,175.157,21.116,153.421
C06679=1085.579,147.413,-68.729,175.155,21.114,153.421
C06680=1085.573,147.164,-68.710,175.152,21.113,153.421
C06681=1085.568,146.915,-68.689,175.150,21.111,153.421
C06682=1085.563,146.666,-68.668,175.148,21.109,153.421
C06683=1085.556,146.416,-68.648,175.146,21.107,153.421
C06684=1085.551,146.167,-68.628,175.144,21.105,153.421
C06685=1085.546,145.918,-68.607,175.141,21.104,153.421
C06686=1085.540,145.670,-68.586,175.139,21.103,153.421
C06687=1085.534,145.421,-68.566,175.137,21.101,153.421
C06688=1085.529,145.172,-68.545,175.135,21.099,153.421
C06689=1085.523,144.922,-68.524,175.132,21.097,153.421
C06690=1085.517,144.673,-68.504,175.131,21.095,153.421
C06691=1085.512,144.424,-68.484,175.128,21.094,153.421
C06692=1085.507,144.175,-68.463,175.126,21.092,153.421
C06693=1085.500,143.896,-68.440,175.123,21.090,153.421
C06694=1085.494,143.617,-68.417,175.121,21.088,153.421
C06695=1085.488,143.338,-68.395,175.118,21.086,153.421
C06696=1085.482,143.060,-68.371,175.116,21.084,153.421
C06697=1085.475,142.811,-68.351,175.114,21.083,153.421
C06698=1085.470,142.562,-68.331,175.111,21.081,153.421
C06699=1085.465,142.312,-68.310,175.109,21.079,153.421
C06700=1085.459,142.064,-68.290,175.107,21.077,153.421
C06701=1085.453,141.814,-68.269,175.105,21.075,153.421
C06702=1085.448,141.565,-68.250,175.103,21.074,153.421
C06703=1085.442,141.316,-68.230,175.100,21.072,153.421
C06704=1085.437,141.067,-68.209,175.098,21.071,153.421
C06705=1085.432,140.818,-68.189,175.096,21.069,153.421
C06706=1085.426,140.569,-68.169,175.094,21.067,153.421
C06707=1085.420,140.319,-68.148,175.092,21.065,153.421
C06708=1085.414,140.070,-68.128,175.090,21.064,153.421
C06709=1085.409,139.821,-68.107,175.087,21.062,153.421
C06710=1085.403,139.572,-68.087,175.085,21.060,153.421
C06711=1085.397,139.323,-68.067,175.083,21.058,153.421
C06712=1085.392,139.074,-68.046,175.081,21.056,153.421
C06713=1085.387,138.825,-68.027,175.079,21.054,153.421
C06714=1085.381,138.575,-68.006,175.076,21.053,153.421
C06715=1085.375,138.327,-67.986,175.075,21.051,153.421
C06716=1085.370,138.078,-67.966,175.072,21.050,153.421
C06717=1085.364,137.829,-67.946,175.070,21.048,153.421
C06718=1085.358,137.580,-67.926,175.068,21.046,153.421
C06719=1085.352,137.329,-67.906,175.066,21.045,153.421
C06720=1085.346,137.081,-67.886,175.063,21.043,153.421
C06721=1085.341,136.832,-67.865,175.061,21.041,153.421
C06722=1085.335,136.583,-67.845,175.059,21.039,153.421
C06723=1085.330,136.333,-67.825,175.057,21.037,153.421
C06724=1085.324,136.084,-67.805,175.055,21.035,153.421
C06725=1085.319,135.835,-67.785,175.053,21.034,153.421
C06726=1085.313,135.586,-67.765,175.051,21.032,153.421
C06727=1085.307,135.337,-67.746,175.048,21.030,153.421
C06728=1085.302,135.088,-67.725,175.046,21.028,153.421
C06729=1085.296,134.839,-67.705,175.044,21.027,153.421
C06730=1085.291,134.590,-67.685,175.042,21.025,153.421
C06731=1085.285,134.340,-67.665,175.040,21.023,153.421
C06732=1085.279,134.092,-67.645,175.038,21.022,153.420
C06733=1085.274,133.842,-67.625,175.036,21.020,153.420
C06734=1085.268,133.593,-67.606,175.033,21.018,153.420
C06735=1085.263,133.344,-67.585,175.031,21.016,153.420
C06736=1085.257,133.094,-67.566,175.029,21.014,153.420
C06737=1085.251,132.846,-67.546,175.027,21.013,153.420
C06738=1085.246,132.596,-67.525,175.025,21.011,153.420
C06739=1085.240,132.347,-67.506,175.023,21.009,153.420
C06740=1085.235,132.098,-67.485,175.021,21.007,153.420
C06741=1085.229,131.849,-67.466,175.018,21.005,153.420
C06742=1085.223,131.600,-67.446,175.017,21.004,153.420
C06743=1085.217,131.351,-67.426,175.014,21.002,153.420
C06744=1085.212,131.101,-67.407,175.012,21.000,153.420
C06745=1085.206,130.852,-67.387,175.010,20.999,153.420
C06746=1085.201,130.603,-67.367,175.008,20.997,153.420
C06747=1085.195,130.354,-67.347,175.006,20.995,153.420
C06748=1085.189,130.105,-67.328,175.004,20.993,153.420
C06749=1085.183,129.856,-67.308,175.002,20.992,153.420
C06750=1085.177,129.606,-67.289,174.999,20.990,153.420
C06751=1085.172,129.357,-67.268,174.997,20.988,153.420
C06752=1085.166,129.108,-67.249,174.995,20.986,153.420
C06753=1085.160,128.859,-67.229,174.993,20.984,153.420
C06754=1085.155,128.610,-67.210,174.991,20.982,153.420
C06755=1085.149,128.361,-67.190,174.989,20.981,153.420
C06756=1085.143,128.111,-67.171,174.987,20.979,153.420
C06757=1085.137,127.833,-67.148,174.984,20.977,153.420
C06758=1085.131,127.554,-67.126,174.982,20.975,153.420
C06759=1085.125,127.274,-67.104,174.980,20.973,153.420
C06760=1085.118,126.996,-67.083,174.977,20.971,153.420
C06761=1085.112,126.747,-67.063,174.976,20.970,153.420
C06762=1085.106,126.498,-67.043,174.973,20.968,153.420
C06763=1085.101,126.248,-67.024,174.971,20.966,153.420
C06764=1085.095,125.999,-67.005,174.970,20.964,153.420
C06765=1085.090,125.750,-66.984,174.967,20.962,153.420
C06766=1085.085,125.501,-66.965,174.965,20.960,153.420
C06767=1085.079,125.252,-66.946,174.963,20.959,153.420
C06768=1085.073,125.003,-66.926,174.961,20.957,153.420
C06769=1085.067,124.754,-66.907,174.958,20.955,153.420
C06770=1085.062,124.504,-66.888,174.957,20.954,153.420
C06771=1085.056,124.255,-66.868,174.955,20.952,153.420
C06772=1085.050,124.006,-66.849,174.952,20.950,153.420
C06773=1085.044,123.756,-66.829,174.951,20.948,153.419
C06774=1085.039,123.508,-66.810,174.948,20.946,153.419
C06775=1085.033,123.259,-66.790,174.946,20.944,153.419
C06776=1085.027,123.009,-66.771,174.945,20.943,153.419
C06777=1085.022,122.760,-66.752,174.942,20.941,153.419
C06778=1085.017,122.511,-66.731,174.940,20.939,153.419
C06779=1085.011,122.261,-66.712,174.938,20.937,153.419
C06780=1085.006,122.013,-66.693,174.936,20.935,153.419
C06781=1085.000,121.763,-66.674,174.934,20.933,153.419
C06782=1084.994,121.514,-66.655,174.932,20.932,153.419
C06783=1084.988,121.265,-66.635,174.930,20.930,153.419
C06784=1084.983,121.016,-66.616,174.928,20.928,153.419
C06785=1084.978,120.767,-66.597,174.926,20.926,153.419
C06786=1084.972,120.517,-66.578,174.924,20.924,153.419
C06787=1084.966,120.268,-66.558,174.922,20.923,153.419
C06788=1084.961,120.019,-66.539,174.920,20.921,153.419
C06789=1084.955,119.770,-66.519,174.917,20.919,153.419
C06790=1084.949,119.521,-66.500,174.916,20.917,153.419
C06791=1084.944,119.272,-66.481,174.914,20.915,153.419
C06792=1084.938,119.022,-66.462,174.911,20.913,153.419
C06793=1084.932,118.773,-66.442,174.910,20.912,153.419
C06794=1084.927,118.524,-66.424,174.908,20.909,153.418
C06795=1084.922,118.275,-66.404,174.906,20.908,153.418
C06796=1084.916,118.025,-66.385,174.904,20.906,153.418
C06797=1084.910,117.776,-66.366,174.901,20.904,153.418
C06798=1084.905,117.527,-66.347,174.900,20.902,153.418
C06799=1084.899,117.278,-66.328,174.898,20.900,153.418
C06800=1084.894,117.028,-66.308,174.895,20.898,153.418
C06801=1084.889,116.779,-66.290,174.894,20.896,153.418
C06802=1084.883,116.530,-66.270,174.892,20.894,153.418
C06803=1084.877,116.280,-66.251,174.890,20.893,153.418
C06804=1084.872,116.032,-66.232,174.888,20.891,153.418
C06805=1084.867,115.782,-66.213,174.885,20.888,153.418
C06806=1084.861,115.533,-66.194,174.884,20.887,153.418
C06807=1084.856,115.284,-66.175,174.882,20.885,153.418
C06808=1084.850,115.035,-66.156,174.880,20.883,153.417
C06809=1084.844,114.785,-66.136,174.878,20.881,153.417
C06810=1084.839,114.537,-66.118,174.875,20.879,153.417
C06811=1084.833,114.287,-66.099,174.874,20.877,153.417
C06812=1084.827,114.038,-66.080,174.872,20.875,153.417
C06813=1084.822,113.789,-66.060,174.869,20.874,153.417
C06814=1084.816,113.540,-66.042,174.868,20.872,153.417
C06815=1084.810,113.291,-66.023,174.866,20.870,153.417
C06816=1084.804,113.041,-66.004,174.864,20.868,153.417
C06817=1084.799,112.793,-65.985,174.862,20.866,153.417
C06818=1084.794,112.543,-65.966,174.860,20.864,153.417
C06819=1084.788,112.293,-65.947,174.858,20.862,153.417
C06820=1084.782,112.045,-65.929,174.856,20.860,153.417
C06821=1084.776,111.765,-65.907,174.854,20.858,153.417
C06822=1084.769,111.486,-65.886,174.851,20.856,153.417
C06823=1084.763,111.207,-65.865,174.850,20.854,153.417
C06824=1084.757,110.928,-65.844,174.847,20.852,153.417
C06825=1084.752,110.680,-65.825,174.845,20.850,153.416
C06826=1084.745,110.430,-65.806,174.843,20.848,153.416
C06827=1084.740,110.180,-65.788,174.841,20.846,153.416
C06828=1084.735,109.932,-65.769,174.839,20.845,153.416
C06829=1084.728,109.683,-65.750,174.837,20.843,153.416
C06830=1084.723,109.433,-65.731,174.835,20.841,153.416
C06831=1084.717,109.185,-65.713,174.834,20.839,153.416
C06832=1084.711,108.935,-65.694,174.831,20.837,153.416
C06833=1084.706,108.685,-65.675,174.829,20.835,153.416
C06834=1084.700,108.437,-65.657,174.828,20.833,153.416
C06835=1084.695,108.187,-65.638,174.825,20.832,153.416
C06836=1084.688,107.938,-65.620,174.824,20.830,153.416
C06837=1084.683,107.689,-65.601,174.822,20.828,153.416
C06838=1084.677,107.439,-65.581,174.820,20.826,153.416
C06839=1084.671,107.190,-65.564,174.818,20.824,153.415
C06840=1084.666,106.941,-65.545,174.816,20.822,153.415
C06841=1084.660,106.692,-65.526,174.814,20.820,153.415
C06842=1084.655,106.442,-65.508,174.812,20.818,153.415
C06843=1084.649,106.193,-65.489,174.810,20.817,153.415
C06844=1084.643,105.943,-65.471,174.808,20.815,153.415
C06845=1084.638,105.695,-65.452,174.806,20.812,153.415
C06846=1084.632,105.445,-65.433,174.804,20.811,153.415
C06847=1084.627,105.196,-65.415,174.802,20.808,153.415
C06848=1084.620,104.947,-65.396,174.801,20.807,153.415
C06849=1084.616,104.698,-65.378,174.798,20.805,153.415
C06850=1084.610,104.448,-65.359,174.797,20.803,153.415
C06851=1084.604,104.199,-65.340,174.795,20.801,153.415
C06852=1084.599,103.950,-65.322,174.793,20.799,153.414
C06853=1084.592,103.701,-65.303,174.791,20.797,153.414
C06854=1084.588,103.451,-65.285,174.789,20.795,153.414
C06855=1084.581,103.202,-65.267,174.787,20.793,153.414
C06856=1084.576,102.953,-65.249,174.785,20.791,153.414
C06857=1084.570,102.704,-65.230,174.783,20.789,153.414
C06858=1084.565,102.454,-65.212,174.781,20.788,153.414
C06859=1084.559,102.205,-65.193,174.780,20.786,153.414
C06860=1084.554,101.956,-65.175,174.777,20.784,153.414
C06861=1084.548,101.706,-65.156,174.775,20.781,153.414
C06862=1084.543,101.457,-65.138,174.774,20.780,153.414
C06863=1084.537,101.208,-65.119,174.772,20.777,153.414
C06864=1084.532,100.959,-65.101,174.770,20.776,153.414
C06865=1084.525,100.710,-65.083,174.768,20.773,153.413
C06866=1084.520,100.460,-65.064,174.766,20.772,153.413
C06867=1084.514,100.211,-65.047,174.764,20.770,153.413
C06868=1084.508,99.962,-65.028,174.763,20.768,153.413
C06869=1084.503,99.712,-65.010,174.760,20.766,153.413
C06870=1084.497,99.463,-64.991,174.759,20.764,153.413
C06871=1084.491,99.214,-64.973,174.757,20.762,153.413
C06872=1084.486,98.964,-64.955,174.754,20.760,153.413
C06873=1084.480,98.716,-64.937,174.753,20.758,153.413
C06874=1084.474,98.466,-64.919,174.751,20.757,153.413
C06875=1084.469,98.217,-64.900,174.749,20.755,153.413
C06876=1084.463,97.967,-64.882,174.747,20.753,153.413
C06877=1084.457,97.718,-64.864,174.746,20.751,153.412
C06878=1084.451,97.469,-64.845,174.743,20.749,153.412
C06879=1084.446,97.220,-64.828,174.742,20.747,153.412
C06880=1084.440,96.970,-64.810,174.739,20.745,153.412
C06881=1084.434,96.722,-64.791,174.738,20.743,153.412
C06882=1084.428,96.472,-64.773,174.736,20.741,153.412
C06883=1084.423,96.223,-64.755,174.734,20.739,153.412
C06884=1084.417,95.974,-64.738,174.732,20.737,153.412
C06885=1084.411,95.695,-64.717,174.730,20.735,153.412
C06886=1084.404,95.415,-64.697,174.728,20.733,153.412
C06887=1084.398,95.136,-64.676,174.726,20.731,153.412
C06888=1084.392,94.858,-64.656,174.724,20.728,153.411
C06889=1084.386,94.608,-64.638,174.722,20.726,153.411
C06890=1084.381,94.359,-64.620,174.720,20.725,153.411
C06891=1084.375,94.110,-64.602,174.718,20.723,153.411
C06892=1084.369,93.861,-64.584,174.717,20.721,153.411
C06893=1084.364,93.612,-64.566,174.715,20.718,153.411
C06894=1084.358,93.362,-64.548,174.713,20.717,153.411
C06895=1084.353,93.113,-64.530,174.711,20.714,153.411
C06896=1084.346,92.863,-64.512,174.709,20.713,153.411
C06897=1084.341,92.614,-64.494,174.707,20.710,153.411
C06898=1084.336,92.365,-64.476,174.705,20.708,153.411
C06899=1084.330,92.115,-64.458,174.704,20.707,153.410
C06900=1084.325,91.866,-64.440,174.701,20.704,153.410
C06901=1084.319,91.617,-64.423,174.700,20.703,153.410
C06902=1084.313,91.368,-64.405,174.698,20.700,153.410
C06903=1084.308,91.119,-64.386,174.696,20.699,153.410
C06904=1084.302,90.869,-64.368,174.694,20.696,153.410
C06905=1084.296,90.620,-64.351,174.693,20.695,153.410
C06906=1084.291,90.371,-64.333,174.690,20.692,153.410
C06907=1084.285,90.121,-64.315,174.689,20.691,153.410
C06908=1084.279,89.872,-64.297,174.687,20.689,153.409
C06909=1084.273,89.622,-64.280,174.685,20.687,153.409
C06910=1084.267,89.373,-64.262,174.683,20.685,153.409
C06911=1084.262,89.124,-64.244,174.682,20.683,153.409
C06912=1084.256,88.875,-64.226,174.679,20.681,153.409
C06913=1084.250,88.626,-64.209,174.678,20.679,153.409
C06914=1084.244,88.376,-64.191,174.676,20.677,153.409
C06915=1084.239,88.127,-64.173,174.674,20.675,153.409
C06916=1084.233,87.878,-64.156,174.672,20.673,153.409
C06917=1084.227,87.628,-64.138,174.671,20.671,153.409
C06918=1084.221,87.379,-64.120,174.669,20.669,153.408
C06919=1084.216,87.130,-64.103,174.667,20.667,153.408
C06920=1084.210,86.880,-64.085,174.665,20.665,153.408
C06921=1084.204,86.631,-64.067,174.663,20.663,153.408
C06922=1084.199,86.382,-64.050,174.661,20.661,153.408
C06923=1084.193,86.132,-64.032,174.660,20.659,153.408
C06924=1084.187,85.883,-64.014,174.658,20.657,153.408
C06925=1084.182,85.634,-63.997,174.656,20.655,153.408
C06926=1084.175,85.385,-63.979,174.654,20.653,153.408
C06927=1084.170,85.135,-63.962,174.653,20.651,153.407
C06928=1084.165,84.886,-63.944,174.650,20.649,153.407
C06929=1084.159,84.636,-63.926,174.649,20.647,153.407
C06930=1084.153,84.387,-63.909,174.647,20.645,153.407
C06931=1084.148,84.138,-63.891,174.645,20.643,153.407
C06932=1084.142,83.889,-63.874,174.643,20.641,153.407
C06933=1084.136,83.639,-63.856,174.642,20.639,153.407
C06934=1084.131,83.390,-63.839,174.639,20.637,153.407
C06935=1084.125,83.141,-63.821,174.638,20.635,153.407
C06936=1084.119,82.891,-63.803,174.637,20.633,153.406
C06937=1084.114,82.642,-63.786,174.634,20.631,153.406
C06938=1084.108,82.393,-63.768,174.633,20.629,153.406
C06939=1084.103,82.144,-63.751,174.631,20.627,153.406
C06940=1084.097,81.893,-63.733,174.630,20.625,153.406
C06941=1084.091,81.644,-63.716,174.627,20.623,153.406
C06942=1084.086,81.395,-63.698,174.626,20.621,153.406
C06943=1084.080,81.146,-63.681,174.624,20.618,153.406
C06944=1084.075,80.897,-63.664,174.622,20.617,153.406
C06945=1084.068,80.647,-63.647,174.620,20.614,153.405
C06946=1084.063,80.398,-63.629,174.619,20.612,153.405
C06947=1084.057,80.149,-63.611,174.617,20.611,153.405
C06948=1084.052,79.899,-63.595,174.615,20.609,153.405
C06949=1084.045,79.620,-63.575,174.613,20.606,153.405
C06950=1084.039,79.342,-63.555,174.611,20.604,153.405
C06951=1084.033,79.063,-63.536,174.609,20.601,153.405
C06952=1084.026,78.784,-63.516,174.607,20.599,153.404
C06953=1084.021,78.534,-63.499,174.605,20.597,153.404
C06954=1084.015,78.285,-63.482,174.604,20.595,153.404
C06955=1084.009,78.036,-63.465,174.602,20.593,153.404
C06956=1084.004,77.786,-63.448,174.600,20.591,153.404
C06957=1083.998,77.537,-63.430,174.598,20.589,153.404
C06958=1083.992,77.288,-63.412,174.597,20.587,153.404
C06959=1083.987,77.039,-63.396,174.595,20.585,153.404
C06960=1083.981,76.790,-63.379,174.593,20.583,153.403
C06961=1083.975,76.539,-63.361,174.592,20.581,153.403
C06962=1083.969,76.291,-63.344,174.590,20.579,153.403
C06963=1083.963,76.041,-63.327,174.588,20.577,153.403
C06964=1083.958,75.792,-63.310,174.586,20.575,153.403
C06965=1083.953,75.543,-63.292,174.585,20.573,153.403
C06966=1083.946,75.293,-63.276,174.582,20.570,153.403
C06967=1083.941,75.044,-63.258,174.581,20.569,153.403
C06968=1083.935,74.794,-63.241,174.579,20.566,153.403
C06969=1083.929,74.545,-63.224,174.578,20.565,153.402
C06970=1083.924,74.296,-63.208,174.575,20.562,153.402
C06971=1083.918,74.047,-63.190,174.574,20.561,153.402
C06972=1083.912,73.797,-63.173,174.573,20.559,153.402
C06973=1083.906,73.548,-63.156,174.570,20.556,153.402
C06974=1083.901,73.298,-63.138,174.569,20.554,153.402
C06975=1083.895,73.049,-63.122,174.567,20.552,153.402
C06976=1083.890,72.799,-63.105,174.565,20.550,153.402
C06977=1083.884,72.550,-63.088,174.563,20.548,153.401
C06978=1083.878,72.301,-63.071,174.562,20.546,153.401
C06979=1083.873,72.052,-63.054,174.560,20.543,153.401
C06980=1083.867,71.802,-63.037,174.558,20.542,153.401
C06981=1083.861,71.553,-63.020,174.557,20.540,153.401
C06982=1083.855,71.303,-63.003,174.555,20.538,153.401
C06983=1083.850,71.054,-62.985,174.554,20.536,153.401
C06984=1083.844,70.805,-62.969,174.551,20.534,153.401
C06985=1083.839,70.555,-62.952,174.550,20.532,153.400
C06986=1083.832,70.307,-62.935,174.548,20.529,153.400
C06987=1083.827,70.057,-62.918,174.547,20.527,153.400
C06988=1083.822,69.808,-62.901,174.544,20.525,153.400
C06989=1083.815,69.558,-62.884,174.543,20.523,153.400
C06990=1083.810,69.308,-62.867,174.542,20.521,153.400
C06991=1083.804,69.059,-62.850,174.539,20.519,153.400
C06992=1083.798,68.810,-62.833,174.538,20.517,153.399
C06993=1083.793,68.560,-62.817,174.536,20.514,153.399
C06994=1083.787,68.311,-62.800,174.534,20.513,153.399
C06995=1083.781,68.062,-62.783,174.532,20.511,153.399
C06996=1083.776,67.812,-62.766,174.531,20.509,153.399
C06997=1083.770,67.564,-62.749,174.530,20.507,153.399
C06998=1083.764,67.314,-62.733,174.528,20.504,153.399
C06999=1083.758,67.065,-62.716,174.526,20.503,153.399
C07000=1083.753,66.815,-62.699,174.524,20.500,153.398
C07001=1083.747,66.566,-62.683,174.523,20.498,153.398
C07002=1083.741,66.316,-62.665,174.521,20.496,153.398
C07003=1083.735,66.066,-62.649,174.519,20.494,153.398
C07004=1083.729,65.817,-62.633,174.518,20.492,153.398
C07005=1083.724,65.568,-62.615,174.516,20.490,153.398
C07006=1083.718,65.319,-62.599,174.514,20.488,153.398
C07007=1083.713,65.069,-62.582,174.512,20.486,153.397
C07008=1083.707,64.820,-62.566,174.511,20.484,153.397
C07009=1083.701,64.570,-62.549,174.509,20.481,153.397
C07010=1083.695,64.321,-62.532,174.507,20.480,153.397
C07011=1083.689,64.072,-62.516,174.506,20.478,153.397
C07012=1083.684,63.822,-62.499,174.504,20.475,153.397
C07013=1083.677,63.544,-62.481,174.502,20.473,153.397
C07014=1083.670,63.265,-62.462,174.500,20.471,153.396
C07015=1083.664,62.986,-62.443,174.498,20.468,153.396
C07016=1083.658,62.707,-62.425,174.496,20.466,153.396
C07017=1083.652,62.457,-62.409,174.495,20.464,153.396
C07018=1083.646,62.208,-62.392,174.493,20.462,153.396
C07019=1083.640,61.959,-62.376,174.491,20.460,153.396
C07020=1083.634,61.710,-62.359,174.490,20.458,153.396
C07021=1083.628,61.460,-62.342,174.488,20.456,153.395
C07022=1083.623,61.211,-62.326,174.486,20.454,153.395
C07023=1083.617,60.961,-62.310,174.485,20.452,153.395
C07024=1083.611,60.712,-62.293,174.483,20.450,153.395
C07025=1083.605,60.462,-62.277,174.481,20.448,153.395
C07026=1083.599,60.213,-62.260,174.479,20.445,153.395
C07027=1083.593,59.964,-62.244,174.478,20.444,153.395
C07028=1083.588,59.714,-62.228,174.476,20.441,153.395
C07029=1083.582,59.465,-62.211,174.474,20.439,153.394
C07030=1083.576,59.215,-62.195,174.473,20.437,153.394
C07031=1083.570,58.966,-62.178,174.471,20.435,153.394
C07032=1083.564,58.717,-62.162,174.469,20.433,153.394
C07033=1083.559,58.467,-62.146,174.467,20.431,153.394
C07034=1083.553,58.218,-62.129,174.466,20.429,153.394
C07035=1083.547,57.968,-62.113,174.465,20.427,153.394
C07036=1083.541,57.719,-62.097,174.463,20.425,153.393
C07037=1083.535,57.470,-62.080,174.461,20.423,153.393
C07038=1083.530,57.220,-62.064,174.459,20.420,153.393
C07039=1083.524,56.971,-62.048,174.458,20.419,153.393
C07040=1083.518,56.721,-62.031,174.456,20.417,153.393
C07041=1083.512,56.472,-62.015,174.454,20.414,153.393
C07042=1083.506,56.223,-61.998,174.453,20.412,153.393
C07043=1083.500,55.973,-61.982,174.452,20.410,153.392
C07044=1083.495,55.724,-61.966,174.450,20.408,153.392
C07045=1083.489,55.475,-61.950,174.448,20.406,153.392
C07046=1083.484,55.224,-61.934,174.446,20.403,153.392
C07047=1083.478,54.976,-61.918,174.445,20.402,153.392
C07048=1083.472,54.726,-61.901,174.443,20.400,153.392
C07049=1083.466,54.477,-61.885,174.441,20.397,153.392
C07050=1083.460,54.228,-61.869,174.440,20.395,153.391
C07051=1083.455,53.978,-61.853,174.438,20.393,153.391
C07052=1083.449,53.729,-61.836,174.436,20.391,153.391
C07053=1083.444,53.479,-61.820,174.435,20.389,153.391
C07054=1083.438,53.229,-61.804,174.433,20.387,153.391
C07055=1083.432,52.980,-61.788,174.432,20.385,153.391
C07056=1083.426,52.731,-61.772,174.430,20.382,153.390
C07057=1083.420,52.482,-61.756,174.428,20.380,153.390
C07058=1083.415,52.232,-61.740,174.427,20.378,153.390
C07059=1083.409,51.983,-61.724,174.425,20.376,153.390
C07060=1083.403,51.733,-61.708,174.423,20.374,153.390
C07061=1083.398,51.484,-61.691,174.422,20.372,153.390
C07062=1083.392,51.234,-61.674,174.420,20.370,153.390
C07063=1083.387,50.985,-61.659,174.419,20.368,153.389
C07064=1083.381,50.736,-61.643,174.417,20.365,153.389
C07065=1083.375,50.486,-61.627,174.415,20.363,153.389
C07066=1083.369,50.237,-61.610,174.414,20.361,153.389
C07067=1083.363,49.987,-61.595,174.412,20.359,153.389
C07068=1083.357,49.738,-61.579,174.411,20.357,153.389
C07069=1083.352,49.489,-61.563,174.409,20.355,153.388
C07070=1083.346,49.239,-61.547,174.407,20.352,153.388
C07071=1083.340,48.990,-61.531,174.406,20.351,153.388
C07072=1083.334,48.740,-61.515,174.404,20.348,153.388
C07073=1083.329,48.490,-61.499,174.402,20.346,153.388
C07074=1083.324,48.241,-61.483,174.401,20.344,153.388
C07075=1083.318,47.992,-61.466,174.399,20.342,153.387
C07076=1083.313,47.742,-61.451,174.398,20.340,153.387
C07077=1083.306,47.463,-61.433,174.396,20.337,153.387
C07078=1083.300,47.184,-61.415,174.394,20.335,153.387
C07079=1083.293,46.905,-61.397,174.392,20.332,153.387
C07080=1083.287,46.626,-61.379,174.390,20.330,153.387
C07081=1083.281,46.376,-61.364,174.389,20.328,153.386
C07082=1083.276,46.128,-61.348,174.388,20.326,153.386
C07083=1083.270,45.878,-61.332,174.386,20.323,153.386
C07084=1083.264,45.628,-61.316,174.384,20.321,153.386
C07085=1083.259,45.378,-61.300,174.382,20.319,153.386
C07086=1083.253,45.130,-61.284,174.381,20.317,153.386
C07087=1083.247,44.880,-61.268,174.380,20.315,153.385
C07088=1083.242,44.630,-61.253,174.377,20.312,153.385
C07089=1083.236,44.382,-61.237,174.376,20.310,153.385
C07090=1083.231,44.132,-61.221,174.375,20.308,153.385
C07091=1083.225,43.882,-61.205,174.373,20.306,153.385
C07092=1083.219,43.632,-61.189,174.372,20.304,153.385
C07093=1083.214,43.384,-61.174,174.370,20.302,153.384
C07094=1083.208,43.134,-61.158,174.368,20.300,153.384
C07095=1083.202,42.884,-61.142,174.367,20.298,153.384
C07096=1083.196,42.635,-61.127,174.365,20.295,153.384
C07097=1083.190,42.386,-61.111,174.363,20.293,153.384
C07098=1083.185,42.136,-61.095,174.362,20.291,153.384
C07099=1083.179,41.887,-61.079,174.360,20.289,153.384
C07100=1083.173,41.637,-61.064,174.359,20.287,153.383
C07101=1083.168,41.388,-61.048,174.357,20.285,153.383
C07102=1083.161,41.138,-61.033,174.355,20.282,153.383
C07103=1083.156,40.888,-61.017,174.354,20.280,153.383
C07104=1083.150,40.640,-61.001,174.353,20.278,153.383
C07105=1083.145,40.390,-60.986,174.351,20.276,153.383
C07106=1083.139,40.141,-60.970,174.349,20.274,153.382
C07107=1083.133,39.892,-60.955,174.348,20.272,153.382
C07108=1083.127,39.642,-60.939,174.346,20.269,153.382
C07109=1083.121,39.392,-60.923,174.345,20.267,153.382
C07110=1083.116,39.143,-60.908,174.343,20.265,153.382
C07111=1083.111,38.893,-60.892,174.341,20.263,153.382
C07112=1083.104,38.644,-60.877,174.340,20.261,153.381
C07113=1083.098,38.394,-60.861,174.339,20.259,153.381
C07114=1083.093,38.145,-60.846,174.337,20.256,153.381
C07115=1083.087,37.895,-60.830,174.335,20.254,153.381
C07116=1083.081,37.646,-60.815,174.333,20.252,153.381
C07117=1083.076,37.396,-60.800,174.332,20.250,153.381
C07118=1083.070,37.147,-60.783,174.331,20.248,153.380
C07119=1083.064,36.897,-60.768,174.329,20.246,153.380
C07120=1083.059,36.648,-60.753,174.327,20.244,153.380
C07121=1083.053,36.399,-60.737,174.326,20.242,153.380
C07122=1083.046,36.149,-60.722,174.324,20.239,153.380
C07123=1083.041,35.900,-60.707,174.323,20.237,153.380
C07124=1083.035,35.650,-60.692,174.321,20.235,153.379
C07125=1083.029,35.401,-60.676,174.319,20.233,153.379
C07126=1083.024,35.152,-60.661,174.318,20.231,153.379
C07127=1083.017,34.902,-60.646,174.317,20.229,153.379
C07128=1083.012,34.652,-60.630,174.314,20.226,153.379
C07129=1083.006,34.403,-60.614,174.313,20.224,153.379
C07130=1083.000,34.154,-60.599,174.312,20.222,153.378
C07131=1082.994,33.904,-60.584,174.310,20.220,153.378
C07132=1082.989,33.655,-60.569,174.309,20.218,153.378
C07133=1082.983,33.405,-60.554,174.307,20.216,153.378
C07134=1082.976,33.156,-60.538,174.305,20.213,153.378
C07135=1082.971,32.907,-60.523,174.304,20.211,153.378
C07136=1082.966,32.657,-60.507,174.303,20.209,153.377
C07137=1082.960,32.408,-60.493,174.301,20.207,153.377
C07138=1082.954,32.158,-60.477,174.299,20.205,153.377
C07139=1082.948,31.908,-60.462,174.298,20.203,153.377
C07140=1082.942,31.659,-60.446,174.297,20.201,153.377
C07141=1082.935,31.380,-60.429,174.295,20.198,153.377
C07142=1082.929,31.101,-60.412,174.293,20.195,153.376
C07143=1082.923,30.822,-60.396,174.291,20.193,153.376
C07144=1082.917,30.543,-60.378,174.289,20.191,153.376
C07145=1082.910,30.293,-60.363,174.288,20.189,153.376
C07146=1082.905,30.044,-60.348,174.287,20.187,153.376
C07147=1082.900,29.794,-60.333,174.285,20.184,153.376
C07148=1082.894,29.545,-60.318,174.283,20.182,153.375
C07149=1082.888,29.295,-60.302,174.282,20.180,153.375
C07150=1082.882,29.045,-60.287,174.280,20.178,153.375
C07151=1082.877,28.796,-60.272,174.279,20.176,153.375
C07152=1082.870,28.546,-60.257,174.277,20.174,153.375
C07153=1082.865,28.297,-60.242,174.275,20.172,153.375
C07154=1082.859,28.048,-60.227,174.274,20.170,153.374
C07155=1082.853,27.799,-60.213,174.273,20.168,153.374
C07156=1082.848,27.549,-60.197,174.271,20.165,153.374
C07157=1082.841,27.299,-60.182,174.269,20.163,153.374
C07158=1082.836,27.050,-60.167,174.268,20.161,153.374
C07159=1082.830,26.800,-60.152,174.266,20.159,153.374
C07160=1082.824,26.551,-60.137,174.265,20.157,153.373
C07161=1082.818,26.301,-60.122,174.263,20.155,153.373
C07162=1082.813,26.052,-60.107,174.262,20.153,153.373
C07163=1082.807,25.802,-60.092,174.260,20.150,153.373
C07164=1082.801,25.553,-60.077,174.259,20.148,153.373
C07165=1082.795,25.304,-60.062,174.257,20.146,153.373
C07166=1082.790,25.054,-60.047,174.255,20.144,153.372
C07167=1082.783,24.805,-60.032,174.254,20.142,153.372
C07168=1082.777,24.555,-60.017,174.253,20.140,153.372
C07169=1082.772,24.306,-60.002,174.251,20.137,153.372
C07170=1082.766,24.055,-59.988,174.249,20.135,153.372
C07171=1082.760,23.807,-59.973,174.248,20.133,153.372
C07172=1082.754,23.557,-59.958,174.246,20.130,153.371
C07173=1082.749,23.308,-59.943,174.245,20.128,153.371
C07174=1082.742,23.058,-59.928,174.244,20.126,153.371
C07175=1082.737,22.809,-59.913,174.242,20.124,153.371
C07176=1082.731,22.559,-59.898,174.240,20.122,153.371
C07177=1082.725,22.310,-59.883,174.239,20.120,153.371
C07178=1082.720,22.059,-59.869,174.238,20.118,153.370
C07179=1082.714,21.810,-59.854,174.236,20.115,153.370
C07180=1082.708,21.562,-59.839,174.234,20.113,153.370
C07181=1082.702,21.312,-59.824,174.233,20.111,153.370
C07182=1082.697,21.063,-59.809,174.231,20.109,153.370
C07183=1082.691,20.812,-59.795,174.230,20.107,153.370
C07184=1082.686,20.563,-59.780,174.228,20.105,153.369
C07185=1082.679,20.313,-59.765,174.227,20.103,153.369
C07186=1082.673,20.064,-59.750,174.225,20.100,153.369
C07187=1082.667,19.815,-59.735,174.224,20.098,153.369
C07188=1082.662,19.565,-59.721,174.223,20.096,153.369
C07189=1082.656,19.315,-59.706,174.220,20.094,153.369
C07190=1082.650,19.066,-59.692,174.219,20.092,153.368
C07191=1082.644,18.816,-59.677,174.218,20.090,153.368
C07192=1082.638,18.567,-59.663,174.217,20.088,153.368
C07193=1082.633,18.318,-59.648,174.214,20.085,153.368
C07194=1082.627,18.068,-59.633,174.213,20.083,153.368
C07195=1082.621,17.819,-59.619,174.212,20.081,153.368
C07196=1082.615,17.569,-59.604,174.210,20.079,153.367
C07197=1082.609,17.320,-59.589,174.209,20.077,153.367
C07198=1082.603,17.070,-59.575,174.207,20.075,153.367
C07199=1082.598,16.820,-59.560,174.206,20.073,153.367
C07200=1082.592,16.571,-59.545,174.204,20.070,153.367
C07201=1082.586,16.321,-59.531,174.203,20.068,153.367
C07202=1082.580,16.072,-59.516,174.201,20.066,153.366
C07203=1082.574,15.823,-59.501,174.199,20.064,153.366
C07204=1082.569,15.573,-59.488,174.198,20.062,153.366
C07205=1082.562,15.295,-59.470,174.197,20.059,153.366
C07206=1082.556,15.017,-59.454,174.195,20.057,153.366
C07207=1082.550,14.740,-59.439,174.194,20.055,153.365
C07208=1082.543,14.462,-59.422,174.191,20.052,153.365
C07209=1082.538,14.213,-59.408,174.190,20.050,153.365
C07210=1082.531,13.963,-59.393,174.188,20.048,153.365
C07211=1082.526,13.713,-59.379,174.187,20.046,153.365
C07212=1082.519,13.464,-59.364,174.186,20.044,153.365
C07213=1082.514,13.214,-59.350,174.184,20.042,153.365
C07214=1082.508,12.965,-59.336,174.182,20.039,153.364
C07215=1082.502,12.716,-59.321,174.181,20.037,153.364
C07216=1082.496,12.466,-59.307,174.180,20.035,153.364
C07217=1082.490,12.216,-59.292,174.178,20.033,153.364
C07218=1082.484,11.967,-59.279,174.176,20.031,153.364
C07219=1082.478,11.718,-59.264,174.175,20.029,153.364
C07220=1082.472,11.468,-59.250,174.174,20.027,153.363
C07221=1082.466,11.219,-59.235,174.172,20.025,153.363
C07222=1082.460,10.969,-59.221,174.170,20.023,153.363
C07223=1082.454,10.720,-59.206,174.169,20.021,153.363
C07224=1082.449,10.470,-59.193,174.168,20.019,153.363
C07225=1082.442,10.220,-59.178,174.166,20.016,153.363
C07226=1082.437,9.971,-59.164,174.164,20.014,153.362
C07227=1082.431,9.721,-59.150,174.163,20.012,153.362
C07228=1082.425,9.472,-59.135,174.162,20.010,153.362
C07229=1082.419,9.222,-59.121,174.160,20.008,153.362
C07230=1082.413,8.972,-59.106,174.159,20.006,153.362
C07231=1082.408,8.723,-59.092,174.157,20.004,153.362
C07232=1082.402,8.474,-59.078,174.156,20.002,153.361
C07233=1082.396,8.224,-59.063,174.154,19.999,153.361
C07234=1082.390,7.974,-59.050,174.153,19.997,153.361
C07235=1082.384,7.725,-59.036,174.151,19.995,153.361
C07236=1082.378,7.476,-59.022,174.150,19.993,153.361
C07237=1082.372,7.226,-59.007,174.148,19.991,153.361
C07238=1082.366,6.977,-58.993,174.147,19.989,153.360
C07239=1082.361,6.727,-58.979,174.145,19.987,153.360
C07240=1082.355,6.477,-58.964,174.144,19.985,153.360
C07241=1082.349,6.228,-58.950,174.142,19.983,153.360
C07242=1082.344,5.978,-58.936,174.141,19.981,153.360
C07243=1082.337,5.729,-58.921,174.139,19.979,153.360
C07244=1082.331,5.479,-58.908,174.137,19.976,153.360
C07245=1082.326,5.230,-58.894,174.136,19.974,153.359
C07246=1082.320,4.981,-58.880,174.135,19.972,153.359
C07247=1082.314,4.730,-58.866,174.133,19.970,153.359
C07248=1082.308,4.481,-58.852,174.131,19.968,153.359
C07249=1082.302,4.232,-58.837,174.130,19.966,153.359
C07250=1082.297,3.982,-58.823,174.129,19.964,153.359
C07251=1082.291,3.732,-58.809,174.128,19.962,153.358
C07252=1082.285,3.483,-58.796,174.126,19.959,153.358
C07253=1082.279,3.234,-58.781,174.124,19.957,153.358
C07254=1082.273,2.984,-58.767,174.123,19.955,153.358
C07255=1082.267,2.734,-58.753,174.122,19.953,153.358
C07256=1082.262,2.484,-58.739,174.120,19.950,153.358
C07257=1082.256,2.236,-58.725,174.119,19.948,153.357
C07258=1082.251,1.986,-58.711,174.117,19.946,153.357
C07259=1082.244,1.736,-58.697,174.116,19.944,153.357
C07260=1082.238,1.486,-58.683,174.114,19.942,153.357
C07261=1082.233,1.237,-58.669,174.113,19.940,153.357
C07262=1082.227,0.988,-58.655,174.111,19.938,153.357
C07263=1082.222,0.738,-58.641,174.110,19.936,153.356
C07264=1082.215,0.488,-58.627,174.108,19.933,153.356
C07265=1082.209,0.239,-58.613,174.107,19.931,153.356
C07266=1082.204,-0.011,-58.600,174.106,19.929,153.356
C07267=1082.198,-0.260,-58.586,174.104,19.927,153.356
C07268=1082.193,-0.510,-58.572,174.103,19.925,153.355
C07269=1082.186,-0.786,-58.557,174.101,19.923,153.355
C07270=1082.180,-1.062,-58.541,174.100,19.921,153.355
C07271=1082.173,-1.337,-58.526,174.098,19.918,153.355
